LIN {X 0,Y 241.734,Z 622.114,A -85,B 0,C 180,E1 -22159.156,E2 -22159.156} C_VEL
LIN {X 0,Y 239.489,Z 637.629,A -85,B 0,C 180,E1 -22159.816,E2 -22159.816} C_VEL
LIN {X 0,Y 236.435,Z 652.725,A -85,B 0,C 180,E1 -22160.765,E2 -22160.765} C_VEL
LIN {X 0,Y 232.635,Z 667.345,A -85,B 0,C 180,E1 -22162.02,E2 -22162.02} C_VEL
LIN {X 0,Y 228.038,Z 681.642,A -85,B 0,C 180,E1 -22163.62,E2 -22163.62} C_VEL
LIN {X 0,Y 222.936,Z 694.986,A -85,B 0,C 180,E1 -22165.531,E2 -22165.531} C_VEL
LIN {X 0,Y 218.006,Z 706.292,A -85,B 0,C 180,E1 -22167.563,E2 -22167.563} C_VEL
LIN {X 0,Y 212.694,Z 717.163,A -85,B 0,C 180,E1 -22169.995,E2 -22169.995} C_VEL
LIN {X 0,Y 207.139,Z 727.482,A -85,B 0,C 180,E1 -22172.879,E2 -22172.879} C_VEL
LIN {X 0,Y 201.494,Z 737.279,A -85,B 0,C 180,E1 -22176.367,E2 -22176.367} C_VEL
LIN {X 0,Y 196.39,Z 745.451,A -85,B 0,C 180,E1 -22180.103,E2 -22180.103} C_VEL
LIN {X 0,Y 192.203,Z 752.008,A -85,B 0,C 180,E1 -22184.008,E2 -22184.008} C_VEL
LIN {X 0,Y 188.734,Z 757.287,A -85,B 0,C 180,E1 -22188.139,E2 -22188.139} C_VEL
LIN {X 0,Y 185.966,Z 761.59,A -85,B 0,C 180,E1 -22192.797,E2 -22192.797} C_VEL
LIN {X 0,Y 184.093,Z 764.533,A -85,B 0,C 180,E1 -22197.694,E2 -22197.694} C_VEL
LIN {X 0,Y 183.006,Z 766.01,A -85,B 0,C 180,E1 -22202.561,E2 -22202.561} C_VEL
LIN {X 0,Y 182.635,Z 766.103,A -85,B 0,C 180,E1 -22207.452,E2 -22207.452} C_VEL
LIN {X 0,Y 182.792,Z 764.903,A -85,B 0,C 180,E1 -22212.088,E2 -22212.088} C_VEL
LIN {X 0,Y 183.127,Z 763.818,A -85,B 0,C 180,E1 -22214.418,E2 -22214.418} C_VEL
LIN {X 0,Y 184.071,Z 760.704,A -85,B 0,C 180,E1 -22218.996,E2 -22218.996} C_VEL
LIN {X 0,Y 185.74,Z 756.271,A -85,B 0,C 180,E1 -22223.483,E2 -22223.483} C_VEL
LIN {X 0,Y 188.123,Z 750.443,A -85,B 0,C 180,E1 -22227.86,E2 -22227.86} C_VEL
LIN {X 0,Y 191.358,Z 743.051,A -85,B 0,C 180,E1 -22232.106,E2 -22232.106} C_VEL
LIN {X 0,Y 194.901,Z 735.115,A -85,B 0,C 180,E1 -22235.692,E2 -22235.692} C_VEL
LIN {X 0,Y 198.898,Z 726.022,A -85,B 0,C 180,E1 -22238.993,E2 -22238.993} C_VEL
LIN {X 0,Y 203.137,Z 715.83,A -85,B 0,C 180,E1 -22241.982,E2 -22241.982} C_VEL
LIN {X 0,Y 207.665,Z 704.233,A -85,B 0,C 180,E1 -22244.705,E2 -22244.705} C_VEL
LIN {X 0,Y 212.179,Z 691.452,A -85,B 0,C 180,E1 -22247.096,E2 -22247.096} C_VEL
LIN {X 0,Y 216.109,Z 678.872,A -85,B 0,C 180,E1 -22248.979,E2 -22248.979} C_VEL
LIN {X 0,Y 219.617,Z 665.333,A -85,B 0,C 180,E1 -22250.611,E2 -22250.611} C_VEL
LIN {X 0,Y 222.901,Z 650.22,A -85,B 0,C 180,E1 -22251.989,E2 -22251.989} C_VEL
LIN {X 0,Y 225.379,Z 635.225,A -85,B 0,C 180,E1 -22253.003,E2 -22253.003} C_VEL
LIN {X 0,Y 227.257,Z 619.581,A -85,B 0,C 180,E1 -22253.706,E2 -22253.706} C_VEL
LIN {X 0,Y 232.606,Z 539.728,A -85,B 0,C 180,E1 -22256.019,E2 -22256.019} C_VEL
LIN {X 0,Y 229.272,Z 532.768,A -85,B 0,C 180,E1 -22257.137,E2 -22257.137} C_VEL
LIN {X 0,Y 222.382,Z 520.492,A -85,B 0,C 180,E1 -22259.498,E2 -22259.498} C_VEL
LIN {X 0,Y 215.018,Z 508.387,A -85,B 0,C 180,E1 -22262.247,E2 -22262.247} C_VEL
LIN {X 0,Y 206.888,Z 496.398,A -85,B 0,C 180,E1 -22265.594,E2 -22265.594} C_VEL
LIN {X 0,Y 200.691,Z 487.945,A -85,B 0,C 180,E1 -22268.442,E2 -22268.442} C_VEL
LIN {X 0,Y 197.937,Z 484.198,A -85,B 0,C 180,E1 -22269.821,E2 -22269.821} C_VEL
LIN {X 0,Y 194.647,Z 480.304,A -85,B 0,C 180,E1 -22271.528,E2 -22271.528} C_VEL
LIN {X 0,Y 193.678,Z 478.802,A -85,B 0,C 180,E1 -22272.082,E2 -22272.082} C_VEL
LIN {X 0,Y 191.056,Z 476.179,A -85,B 0,C 180,E1 -22273.545,E2 -22273.545} C_VEL
LIN {X 0,Y 189.711,Z 473.644,A -85,B 0,C 180,E1 -22274.429,E2 -22274.429} C_VEL
LIN {X 0,Y 187.18,Z 471.799,A -85,B 0,C 180,E1 -22275.917,E2 -22275.917} C_VEL
LIN {X 0,Y 185.806,Z 469.34,A -85,B 0,C 180,E1 -22276.897,E2 -22276.897} C_VEL
LIN {X 0,Y 185.502,Z 467.989,A -85,B 0,C 180,E1 -22277.235,E2 -22277.235} C_VEL
LIN {X 0,Y 185.52,Z 467.989,A -85,B 0,C 180,E1 -22279.908,E2 -22279.908} C_VEL
LIN {X 0,Y 185.547,Z 467.982,A -85,B 0,C 180,E1 -22282.696,E2 -22282.696} C_VEL
LIN {X 0,Y 185.544,Z 467.991,A -85,B 0,C 180,E1 -22287.974,E2 -22287.974} C_VEL
LIN {X 0,Y 185.584,Z 467.969,A -85,B 0,C 180,E1 -22290.577,E2 -22290.577} C_VEL
LIN {X 0,Y 185.583,Z 467.972,A -85,B 0,C 180,E1 -22295.381,E2 -22295.381} C_VEL
LIN {X 0,Y 185.677,Z 467.972,A -85,B 0,C 180,E1 -22301.133,E2 -22301.133} C_VEL
LIN {X 0,Y 185.768,Z 467.969,A -85,B 0,C 180,E1 -22306.879,E2 -22306.879} C_VEL
LIN {X 0,Y 186.017,Z 467.914,A -85,B 0,C 180,E1 -22311.307,E2 -22311.307} C_VEL
LIN {X 0,Y 186.21,Z 467.89,A -85,B 0,C 180,E1 -22317.836,E2 -22317.836} C_VEL
LIN {X 0,Y 186.409,Z 467.888,A -85,B 0,C 180,E1 -22319.999,E2 -22319.999} C_VEL
LIN {X 0,Y 185.926,Z 467.912,A -85,B 0,C 180,E1 -22324.335,E2 -22324.335} C_VEL
LIN {X 0,Y 186.016,Z 467.939,A -85,B 0,C 180,E1 -22328.692,E2 -22328.692} C_VEL
LIN {X 0,Y 185.737,Z 467.946,A -85,B 0,C 180,E1 -22333.122,E2 -22333.122} C_VEL
LIN {X 0,Y 185.72,Z 467.953,A -85,B 0,C 180,E1 -22337.621,E2 -22337.621} C_VEL
LIN {X 0,Y 185.652,Z 468.142,A -85,B 0,C 180,E1 -22340.497,E2 -22340.497} C_VEL
LIN {X 0,Y 186.512,Z 470.625,A -85,B 0,C 180,E1 -22341.192,E2 -22341.192} C_VEL
LIN {X 0,Y 188.316,Z 472.728,A -85,B 0,C 180,E1 -22342.346,E2 -22342.346} C_VEL
LIN {X 0,Y 190.035,Z 473.955,A -85,B 0,C 180,E1 -22343.353,E2 -22343.353} C_VEL
LIN {X 0,Y 191.815,Z 477.044,A -85,B 0,C 180,E1 -22344.486,E2 -22344.486} C_VEL
LIN {X 0,Y 194.264,Z 479.432,A -85,B 0,C 180,E1 -22345.825,E2 -22345.825} C_VEL
LIN {X 0,Y 196.595,Z 482.776,A -85,B 0,C 180,E1 -22347.098,E2 -22347.098} C_VEL
LIN {X 0,Y 198.231,Z 484.658,A -85,B 0,C 180,E1 -22347.919,E2 -22347.919} C_VEL
LIN {X 0,Y 201.912,Z 489.596,A -85,B 0,C 180,E1 -22349.729,E2 -22349.729} C_VEL
LIN {X 0,Y 206.916,Z 496.507,A -85,B 0,C 180,E1 -22352.012,E2 -22352.012} C_VEL
LIN {X 0,Y 213.331,Z 507.607,A -85,B 0,C 180,E1 -22354.774,E2 -22354.774} C_VEL
LIN {X 0,Y 220.542,Z 521.142,A -85,B 0,C 180,E1 -22357.615,E2 -22357.615} C_VEL
LIN {X 0,Y 227.101,Z 535.188,A -85,B 0,C 180,E1 -22360.024,E2 -22360.024} C_VEL
LIN {X 0,Y 231.364,Z 545.348,A -85,B 0,C 180,E1 -22361.526,E2 -22361.526} C_VEL
LIN {X 0,Y 231.715,Z 547.693,A -85,B 0,C 180,E1 -22361.713,E2 -22361.713} C_VEL
LIN {X 0,Y 231.08,Z 551.504,A -85,B 0,C 180,E1 -22361.731,E2 -22361.731} C_VEL
LIN {X 0,Y 229.684,Z 555.211,A -85,B 0,C 180,E1 -22361.564,E2 -22361.564} C_VEL
LIN {X 0,Y 226.875,Z 561.739,A -85,B 0,C 180,E1 -22361.18,E2 -22361.18} C_VEL
LIN {X 0,Y 225.979,Z 565.9,A -85,B 0,C 180,E1 -22361.151,E2 -22361.151} C_VEL
LIN {X 0,Y 221.35,Z 631.555,A -85,B 0,C 180,E1 -22363.091,E2 -22363.091} C_VEL
LIN {X 0,Y 219.258,Z 647.344,A -85,B 0,C 180,E1 -22363.845,E2 -22363.845} C_VEL
LIN {X 0,Y 216.358,Z 662.488,A -85,B 0,C 180,E1 -22364.883,E2 -22364.883} C_VEL
LIN {X 0,Y 213.032,Z 676.219,A -85,B 0,C 180,E1 -22366.147,E2 -22366.147} C_VEL
LIN {X 0,Y 209.192,Z 689.735,A -85,B 0,C 180,E1 -22367.784,E2 -22367.784} C_VEL
LIN {X 0,Y 204.553,Z 703.482,A -85,B 0,C 180,E1 -22369.893,E2 -22369.893} C_VEL
LIN {X 0,Y 199.88,Z 715.958,A -85,B 0,C 180,E1 -22372.343,E2 -22372.343} C_VEL
LIN {X 0,Y 194.715,Z 728.142,A -85,B 0,C 180,E1 -22375.355,E2 -22375.355} C_VEL
LIN {X 0,Y 190.501,Z 737.849,A -85,B 0,C 180,E1 -22378.384,E2 -22378.384} C_VEL
LIN {X 0,Y 186.487,Z 746.873,A -85,B 0,C 180,E1 -22381.895,E2 -22381.895} C_VEL
LIN {X 0,Y 182.942,Z 754.535,A -85,B 0,C 180,E1 -22385.607,E2 -22385.607} C_VEL
LIN {X 0,Y 180.179,Z 760.857,A -85,B 0,C 180,E1 -22389.447,E2 -22389.447} C_VEL
LIN {X 0,Y 177.951,Z 766.646,A -85,B 0,C 180,E1 -22393.95,E2 -22393.95} C_VEL
LIN {X 0,Y 176.573,Z 771.032,A -85,B 0,C 180,E1 -22398.52,E2 -22398.52} C_VEL
LIN {X 0,Y 176.011,Z 774.126,A -85,B 0,C 180,E1 -22403.119,E2 -22403.119} C_VEL
LIN {X 0,Y 175.948,Z 775.99,A -85,B 0,C 180,E1 -22407.71,E2 -22407.71} C_VEL
LIN {X 0,Y 176.088,Z 776.458,A -85,B 0,C 180,E1 -22409.999,E2 -22409.999} C_VEL
LIN {X 0,Y 175.93,Z 776.478,A -85,B 0,C 180,E1 -22414.581,E2 -22414.581} C_VEL
LIN {X 0,Y 176.219,Z 775.363,A -85,B 0,C 180,E1 -22419.178,E2 -22419.178} C_VEL
LIN {X 0,Y 177.172,Z 773.116,A -85,B 0,C 180,E1 -22423.767,E2 -22423.767} C_VEL
LIN {X 0,Y 179.099,Z 769.707,A -85,B 0,C 180,E1 -22428.294,E2 -22428.294} C_VEL
LIN {X 0,Y 181.995,Z 765.027,A -85,B 0,C 180,E1 -22432.714,E2 -22432.714} C_VEL
LIN {X 0,Y 185.858,Z 758.973,A -85,B 0,C 180,E1 -22436.984,E2 -22436.984} C_VEL
LIN {X 0,Y 190.198,Z 752.43,A -85,B 0,C 180,E1 -22440.534,E2 -22440.534} C_VEL
LIN {X 0,Y 195.326,Z 743.996,A -85,B 0,C 180,E1 -22444.217,E2 -22444.217} C_VEL
LIN {X 0,Y 200.526,Z 735.309,A -85,B 0,C 180,E1 -22447.196,E2 -22447.196} C_VEL
LIN {X 0,Y 206.805,Z 724.104,A -85,B 0,C 180,E1 -22450.216,E2 -22450.216} C_VEL
LIN {X 0,Y 212.592,Z 712.612,A -85,B 0,C 180,E1 -22452.662,E2 -22452.662} C_VEL
LIN {X 0,Y 218.333,Z 699.772,A -85,B 0,C 180,E1 -22454.817,E2 -22454.817} C_VEL
LIN {X 0,Y 223.651,Z 686.095,A -85,B 0,C 180,E1 -22456.606,E2 -22456.606} C_VEL
LIN {X 0,Y 228.157,Z 672.417,A -85,B 0,C 180,E1 -22457.997,E2 -22457.997} C_VEL
LIN {X 0,Y 231.692,Z 659.718,A -85,B 0,C 180,E1 -22458.983,E2 -22458.983} C_VEL
LIN {X 0,Y 235.025,Z 644.454,A -85,B 0,C 180,E1 -22459.851,E2 -22459.851} C_VEL
LIN {X 0,Y 237.229,Z 629.636,A -85,B 0,C 180,E1 -22460.465,E2 -22460.465} C_VEL
LIN {X 0,Y 243.268,Z 558.028,A -85,B 0,C 180,E1 -22462.41,E2 -22462.41} C_VEL
LIN {X 0,Y 241.558,Z 553.044,A -85,B 0,C 180,E1 -22463.369,E2 -22463.369} C_VEL
LIN {X 0,Y 237.978,Z 544.448,A -85,B 0,C 180,E1 -22465.447,E2 -22465.447} C_VEL
LIN {X 0,Y 234.157,Z 536.255,A -85,B 0,C 180,E1 -22467.872,E2 -22467.872} C_VEL
LIN {X 0,Y 230.657,Z 529.337,A -85,B 0,C 180,E1 -22470.376,E2 -22470.376} C_VEL
LIN {X 0,Y 228.094,Z 524.709,A -85,B 0,C 180,E1 -22472.473,E2 -22472.473} C_VEL
LIN {X 0,Y 225.797,Z 520.619,A -85,B 0,C 180,E1 -22474.627,E2 -22474.627} C_VEL
LIN {X 0,Y 223.343,Z 517.052,A -85,B 0,C 180,E1 -22477.295,E2 -22477.295} C_VEL
LIN {X 0,Y 222.418,Z 516.005,A -85,B 0,C 180,E1 -22478.45,E2 -22478.45} C_VEL
LIN {X 0,Y 220.305,Z 512.836,A -85,B 0,C 180,E1 -22481.921,E2 -22481.921} C_VEL
LIN {X 0,Y 219.775,Z 511.515,A -85,B 0,C 180,E1 -22483.274,E2 -22483.274} C_VEL
LIN {X 0,Y 218.477,Z 510.721,A -85,B 0,C 180,E1 -22488.872,E2 -22488.872} C_VEL
LIN {X 0,Y 219.031,Z 510.958,A -85,B 0,C 180,E1 -22493.09,E2 -22493.09} C_VEL
LIN {X 0,Y 220.41,Z 511.803,A -85,B 0,C 180,E1 -22496.486,E2 -22496.486} C_VEL
LIN {X 0,Y 222.476,Z 515.52,A -85,B 0,C 180,E1 -22500,E2 -22500} C_VEL
LIN {X 0,Y 223.564,Z 516.901,A -85,B 0,C 180,E1 -22501.369,E2 -22501.369} C_VEL
LIN {X 0,Y 226.489,Z 521.275,A -85,B 0,C 180,E1 -22504.464,E2 -22504.464} C_VEL
LIN {X 0,Y 229.47,Z 526.02,A -85,B 0,C 180,E1 -22507.037,E2 -22507.037} C_VEL
LIN {X 0,Y 232.882,Z 531.325,A -85,B 0,C 180,E1 -22509.526,E2 -22509.526} C_VEL
LIN {X 0,Y 237.163,Z 538.709,A -85,B 0,C 180,E1 -22512.255,E2 -22512.255} C_VEL
LIN {X 0,Y 242.095,Z 547.889,A -85,B 0,C 180,E1 -22514.992,E2 -22514.992} C_VEL
LIN {X 0,Y 243.679,Z 551.454,A -85,B 0,C 180,E1 -22515.825,E2 -22515.825} C_VEL
LIN {X 0,Y 237.763,Z 621.792,A -85,B 0,C 180,E1 -22517.744,E2 -22517.744} C_VEL
LIN {X 0,Y 235.49,Z 637.313,A -85,B 0,C 180,E1 -22518.392,E2 -22518.392} C_VEL
LIN {X 0,Y 232.244,Z 652.905,A -85,B 0,C 180,E1 -22519.362,E2 -22519.362} C_VEL
LIN {X 0,Y 228.145,Z 667.998,A -85,B 0,C 180,E1 -22520.663,E2 -22520.663} C_VEL
LIN {X 0,Y 223.752,Z 681.221,A -85,B 0,C 180,E1 -22522.143,E2 -22522.143} C_VEL
LIN {X 0,Y 218.408,Z 694.763,A -85,B 0,C 180,E1 -22524.072,E2 -22524.072} C_VEL
LIN {X 0,Y 213.217,Z 706.192,A -85,B 0,C 180,E1 -22526.121,E2 -22526.121} C_VEL
LIN {X 0,Y 207.861,Z 716.722,A -85,B 0,C 180,E1 -22528.471,E2 -22528.471} C_VEL
LIN {X 0,Y 201.824,Z 727.5,A -85,B 0,C 180,E1 -22531.49,E2 -22531.49} C_VEL
LIN {X 0,Y 196.463,Z 736.323,A -85,B 0,C 180,E1 -22534.64,E2 -22534.64} C_VEL
LIN {X 0,Y 191.661,Z 743.7,A -85,B 0,C 180,E1 -22537.935,E2 -22537.935} C_VEL
LIN {X 0,Y 187.467,Z 749.95,A -85,B 0,C 180,E1 -22541.431,E2 -22541.431} C_VEL
LIN {X 0,Y 183.952,Z 755.015,A -85,B 0,C 180,E1 -22545.027,E2 -22545.027} C_VEL
LIN {X 0,Y 180.326,Z 760.213,A -85,B 0,C 180,E1 -22549.981,E2 -22549.981} C_VEL
LIN {X 0,Y 178.38,Z 762.986,A -85,B 0,C 180,E1 -22553.775,E2 -22553.775} C_VEL
LIN {X 0,Y 176.639,Z 765.401,A -85,B 0,C 180,E1 -22558.855,E2 -22558.855} C_VEL
LIN {X 0,Y 175.71,Z 766.396,A -85,B 0,C 180,E1 -22563.9,E2 -22563.9} C_VEL
LIN {X 0,Y 175.528,Z 766.041,A -85,B 0,C 180,E1 -22568.88,E2 -22568.88} C_VEL
LIN {X 0,Y 175.898,Z 764.397,A -85,B 0,C 180,E1 -22573.76,E2 -22573.76} C_VEL
LIN {X 0,Y 176.826,Z 761.484,A -85,B 0,C 180,E1 -22578.539,E2 -22578.539} C_VEL
LIN {X 0,Y 178.464,Z 757.262,A -85,B 0,C 180,E1 -22583.216,E2 -22583.216} C_VEL
LIN {X 0,Y 180.846,Z 751.658,A -85,B 0,C 180,E1 -22587.774,E2 -22587.774} C_VEL
LIN {X 0,Y 184.124,Z 744.508,A -85,B 0,C 180,E1 -22592.189,E2 -22592.189} C_VEL
LIN {X 0,Y 187.675,Z 736.853,A -85,B 0,C 180,E1 -22595.912,E2 -22595.912} C_VEL
LIN {X 0,Y 192.068,Z 727.393,A -85,B 0,C 180,E1 -22599.549,E2 -22599.549} C_VEL
LIN {X 0,Y 196.845,Z 716.415,A -85,B 0,C 180,E1 -22602.895,E2 -22602.895} C_VEL
LIN {X 0,Y 201.511,Z 704.901,A -85,B 0,C 180,E1 -22605.683,E2 -22605.683} C_VEL
LIN {X 0,Y 206.186,Z 692.282,A -85,B 0,C 180,E1 -22608.105,E2 -22608.105} C_VEL
LIN {X 0,Y 210.248,Z 679.75,A -85,B 0,C 180,E1 -22610.038,E2 -22610.038} C_VEL
LIN {X 0,Y 213.892,Z 666.336,A -85,B 0,C 180,E1 -22611.695,E2 -22611.695} C_VEL
LIN {X 0,Y 217.262,Z 651.491,A -85,B 0,C 180,E1 -22613.094,E2 -22613.094} C_VEL
LIN {X 0,Y 219.947,Z 636.009,A -85,B 0,C 180,E1 -22614.168,E2 -22614.168} C_VEL
LIN {X 0,Y 221.826,Z 621.311,A -85,B 0,C 180,E1 -22614.858,E2 -22614.858} C_VEL
LIN {X 0,Y 227.367,Z 542.121,A -85,B 0,C 180,E1 -22617.179,E2 -22617.179} C_VEL
LIN {X 0,Y 221.677,Z 531.086,A -85,B 0,C 180,E1 -22619.174,E2 -22619.174} C_VEL
LIN {X 0,Y 212.987,Z 516.086,A -85,B 0,C 180,E1 -22622.465,E2 -22622.465} C_VEL
LIN {X 0,Y 205.507,Z 504.756,A -85,B 0,C 180,E1 -22625.595,E2 -22625.595} C_VEL
LIN {X 0,Y 200.107,Z 497.094,A -85,B 0,C 180,E1 -22628.09,E2 -22628.09} C_VEL
LIN {X 0,Y 197.355,Z 493.344,A -85,B 0,C 180,E1 -22629.459,E2 -22629.459} C_VEL
LIN {X 0,Y 194.47,Z 489.422,A -85,B 0,C 180,E1 -22630.968,E2 -22630.968} C_VEL
LIN {X 0,Y 191.496,Z 485.498,A -85,B 0,C 180,E1 -22632.629,E2 -22632.629} C_VEL
LIN {X 0,Y 188.184,Z 481.692,A -85,B 0,C 180,E1 -22634.588,E2 -22634.588} C_VEL
LIN {X 0,Y 186.961,Z 479.881,A -85,B 0,C 180,E1 -22635.378,E2 -22635.378} C_VEL
LIN {X 0,Y 184.461,Z 477.453,A -85,B 0,C 180,E1 -22636.981,E2 -22636.981} C_VEL
LIN {X 0,Y 182.959,Z 474.622,A -85,B 0,C 180,E1 -22638.13,E2 -22638.13} C_VEL
LIN {X 0,Y 180.327,Z 472.837,A -85,B 0,C 180,E1 -22639.978,E2 -22639.978} C_VEL
LIN {X 0,Y 178.868,Z 470.544,A -85,B 0,C 180,E1 -22641.2,E2 -22641.2} C_VEL
LIN {X 0,Y 178.466,Z 468.876,A -85,B 0,C 180,E1 -22641.703,E2 -22641.703} C_VEL
LIN {X 0,Y 178.492,Z 468.874,A -85,B 0,C 180,E1 -22646.547,E2 -22646.547} C_VEL
LIN {X 0,Y 178.525,Z 468.848,A -85,B 0,C 180,E1 -22650.007,E2 -22650.007} C_VEL
LIN {X 0,Y 178.523,Z 468.856,A -85,B 0,C 180,E1 -22654.886,E2 -22654.886} C_VEL
LIN {X 0,Y 178.625,Z 468.854,A -85,B 0,C 180,E1 -22660.785,E2 -22660.785} C_VEL
LIN {X 0,Y 178.685,Z 468.849,A -85,B 0,C 180,E1 -22666.349,E2 -22666.349} C_VEL
LIN {X 0,Y 178.966,Z 468.79,A -85,B 0,C 180,E1 -22670.962,E2 -22670.962} C_VEL
LIN {X 0,Y 179.156,Z 468.767,A -85,B 0,C 180,E1 -22677.751,E2 -22677.751} C_VEL
LIN {X 0,Y 179.372,Z 468.764,A -85,B 0,C 180,E1 -22679.999,E2 -22679.999} C_VEL
LIN {X 0,Y 178.874,Z 468.79,A -85,B 0,C 180,E1 -22684.506,E2 -22684.506} C_VEL
LIN {X 0,Y 178.966,Z 468.813,A -85,B 0,C 180,E1 -22689.037,E2 -22689.037} C_VEL
LIN {X 0,Y 178.67,Z 468.831,A -85,B 0,C 180,E1 -22693.651,E2 -22693.651} C_VEL
LIN {X 0,Y 178.66,Z 468.886,A -85,B 0,C 180,E1 -22696.056,E2 -22696.056} C_VEL
LIN {X 0,Y 179.368,Z 471.182,A -85,B 0,C 180,E1 -22696.796,E2 -22696.796} C_VEL
LIN {X 0,Y 181.346,Z 473.561,A -85,B 0,C 180,E1 -22698.357,E2 -22698.357} C_VEL
LIN {X 0,Y 183.205,Z 474.802,A -85,B 0,C 180,E1 -22699.631,E2 -22699.631} C_VEL
LIN {X 0,Y 184.787,Z 477.743,A -85,B 0,C 180,E1 -22700.816,E2 -22700.816} C_VEL
LIN {X 0,Y 187.588,Z 480.382,A -85,B 0,C 180,E1 -22702.571,E2 -22702.571} C_VEL
LIN {X 0,Y 189.993,Z 483.914,A -85,B 0,C 180,E1 -22704.1,E2 -22704.1} C_VEL
LIN {X 0,Y 191.71,Z 485.705,A -85,B 0,C 180,E1 -22705.077,E2 -22705.077} C_VEL
LIN {X 0,Y 194.528,Z 489.448,A -85,B 0,C 180,E1 -22706.647,E2 -22706.647} C_VEL
LIN {X 0,Y 199.16,Z 495.74,A -85,B 0,C 180,E1 -22709.026,E2 -22709.026} C_VEL
LIN {X 0,Y 203.688,Z 502.029,A -85,B 0,C 180,E1 -22711.168,E2 -22711.168} C_VEL
LIN {X 0,Y 211.32,Z 515.671,A -85,B 0,C 180,E1 -22714.573,E2 -22714.573} C_VEL
LIN {X 0,Y 217.721,Z 528.372,A -85,B 0,C 180,E1 -22717.173,E2 -22717.173} C_VEL
LIN {X 0,Y 224.288,Z 543.054,A -85,B 0,C 180,E1 -22719.675,E2 -22719.675} C_VEL
LIN {X 0,Y 227.042,Z 550.077,A -85,B 0,C 180,E1 -22720.69,E2 -22720.69} C_VEL
LIN {X 0,Y 225.979,Z 565.9,A -85,B 0,C 180,E1 -22721.151,E2 -22721.151} C_VEL
LIN {X 0,Y 225.101,Z 571.739,A -85,B 0,C 180,E1 -22721.204,E2 -22721.204} C_VEL
LIN {X 0,Y 219.653,Z 590.729,A -85,B 0,C 180,E1 -22720.734,E2 -22720.734} C_VEL
LIN {X 0,Y 218.743,Z 596.569,A -85,B 0,C 180,E1 -22720.779,E2 -22720.779} C_VEL
LIN {X 0,Y 216.099,Z 631.564,A -85,B 0,C 180,E1 -22721.844,E2 -22721.844} C_VEL
LIN {X 0,Y 213.948,Z 647.286,A -85,B 0,C 180,E1 -22722.605,E2 -22722.605} C_VEL
LIN {X 0,Y 211.081,Z 661.823,A -85,B 0,C 180,E1 -22723.599,E2 -22723.599} C_VEL
LIN {X 0,Y 207.356,Z 676.746,A -85,B 0,C 180,E1 -22725,E2 -22725} C_VEL
LIN {X 0,Y 203.517,Z 689.744,A -85,B 0,C 180,E1 -22726.6,E2 -22726.6} C_VEL
LIN {X 0,Y 198.649,Z 703.658,A -85,B 0,C 180,E1 -22728.781,E2 -22728.781} C_VEL
LIN {X 0,Y 193.814,Z 716.078,A -85,B 0,C 180,E1 -22731.279,E2 -22731.279} C_VEL
LIN {X 0,Y 188.845,Z 727.381,A -85,B 0,C 180,E1 -22734.115,E2 -22734.115} C_VEL
LIN {X 0,Y 184.524,Z 736.717,A -85,B 0,C 180,E1 -22737.052,E2 -22737.052} C_VEL
LIN {X 0,Y 180.796,Z 745.008,A -85,B 0,C 180,E1 -22740.288,E2 -22740.288} C_VEL
LIN {X 0,Y 176.882,Z 752.971,A -85,B 0,C 180,E1 -22744.082,E2 -22744.082} C_VEL
LIN {X 0,Y 173.452,Z 760.391,A -85,B 0,C 180,E1 -22748.612,E2 -22748.612} C_VEL
LIN {X 0,Y 171.074,Z 766.242,A -85,B 0,C 180,E1 -22753.286,E2 -22753.286} C_VEL
LIN {X 0,Y 169.569,Z 770.683,A -85,B 0,C 180,E1 -22758.039,E2 -22758.039} C_VEL
LIN {X 0,Y 168.93,Z 773.83,A -85,B 0,C 180,E1 -22762.829,E2 -22762.829} C_VEL
LIN {X 0,Y 168.857,Z 775.732,A -85,B 0,C 180,E1 -22767.613,E2 -22767.613} C_VEL
LIN {X 0,Y 168.996,Z 776.213,A -85,B 0,C 180,E1 -22769.999,E2 -22769.999} C_VEL
LIN {X 0,Y 168.845,Z 776.282,A -85,B 0,C 180,E1 -22774.774,E2 -22774.774} C_VEL
LIN {X 0,Y 169.158,Z 775.22,A -85,B 0,C 180,E1 -22779.565,E2 -22779.565} C_VEL
LIN {X 0,Y 170.221,Z 773.029,A -85,B 0,C 180,E1 -22784.341,E2 -22784.341} C_VEL
LIN {X 0,Y 172.317,Z 769.67,A -85,B 0,C 180,E1 -22789.042,E2 -22789.042} C_VEL
LIN {X 0,Y 175.414,Z 765.026,A -85,B 0,C 180,E1 -22793.617,E2 -22793.617} C_VEL
LIN {X 0,Y 179.519,Z 759.048,A -85,B 0,C 180,E1 -22798.019,E2 -22798.019} C_VEL
LIN {X 0,Y 184.762,Z 751.584,A -85,B 0,C 180,E1 -22802.175,E2 -22802.175} C_VEL
LIN {X 0,Y 190.014,Z 743.452,A -85,B 0,C 180,E1 -22805.733,E2 -22805.733} C_VEL
LIN {X 0,Y 195.813,Z 734.172,A -85,B 0,C 180,E1 -22808.908,E2 -22808.908} C_VEL
LIN {X 0,Y 201.459,Z 724.554,A -85,B 0,C 180,E1 -22811.514,E2 -22811.514} C_VEL
LIN {X 0,Y 207.455,Z 713.229,A -85,B 0,C 180,E1 -22813.984,E2 -22813.984} C_VEL
LIN {X 0,Y 213.354,Z 700.704,A -85,B 0,C 180,E1 -22816.134,E2 -22816.134} C_VEL
LIN {X 0,Y 218.886,Z 687.172,A -85,B 0,C 180,E1 -22817.942,E2 -22817.942} C_VEL
LIN {X 0,Y 223.521,Z 673.816,A -85,B 0,C 180,E1 -22819.334,E2 -22819.334} C_VEL
LIN {X 0,Y 227.466,Z 660.311,A -85,B 0,C 180,E1 -22820.396,E2 -22820.396} C_VEL
LIN {X 0,Y 231.045,Z 644.523,A -85,B 0,C 180,E1 -22821.297,E2 -22821.297} C_VEL
LIN {X 0,Y 233.41,Z 629.037,A -85,B 0,C 180,E1 -22821.929,E2 -22821.929} C_VEL
LIN {X 0,Y 239.383,Z 561.006,A -85,B 0,C 180,E1 -22823.769,E2 -22823.769} C_VEL
LIN {X 0,Y 238.903,Z 559.062,A -85,B 0,C 180,E1 -22824.093,E2 -22824.093} C_VEL
LIN {X 0,Y 235.248,Z 549.883,A -85,B 0,C 180,E1 -22826.335,E2 -22826.335} C_VEL
LIN {X 0,Y 231.652,Z 541.788,A -85,B 0,C 180,E1 -22828.788,E2 -22828.788} C_VEL
LIN {X 0,Y 228.565,Z 535.35,A -85,B 0,C 180,E1 -22831.162,E2 -22831.162} C_VEL
LIN {X 0,Y 226.277,Z 531.044,A -85,B 0,C 180,E1 -22833.141,E2 -22833.141} C_VEL
LIN {X 0,Y 224.362,Z 527.366,A -85,B 0,C 180,E1 -22835.057,E2 -22835.057} C_VEL
LIN {X 0,Y 221.879,Z 523.581,A -85,B 0,C 180,E1 -22837.906,E2 -22837.906} C_VEL
LIN {X 0,Y 219.223,Z 519.836,A -85,B 0,C 180,E1 -22842.194,E2 -22842.194} C_VEL
LIN {X 0,Y 218.753,Z 518.515,A -85,B 0,C 180,E1 -22843.488,E2 -22843.488} C_VEL
LIN {X 0,Y 217.555,Z 517.765,A -85,B 0,C 180,E1 -22848.824,E2 -22848.824} C_VEL
LIN {X 0,Y 218.06,Z 517.969,A -85,B 0,C 180,E1 -22852.933,E2 -22852.933} C_VEL
LIN {X 0,Y 219.307,Z 518.765,A -85,B 0,C 180,E1 -22856.156,E2 -22856.156} C_VEL
LIN {X 0,Y 221.273,Z 522.4,A -85,B 0,C 180,E1 -22859.671,E2 -22859.671} C_VEL
LIN {X 0,Y 222.261,Z 523.81,A -85,B 0,C 180,E1 -22861.001,E2 -22861.001} C_VEL
LIN {X 0,Y 224.909,Z 527.891,A -85,B 0,C 180,E1 -22863.923,E2 -22863.923} C_VEL
LIN {X 0,Y 227.68,Z 532.492,A -85,B 0,C 180,E1 -22866.447,E2 -22866.447} C_VEL
LIN {X 0,Y 231.04,Z 537.931,A -85,B 0,C 180,E1 -22869.025,E2 -22869.025} C_VEL
LIN {X 0,Y 235.185,Z 545.538,A -85,B 0,C 180,E1 -22871.792,E2 -22871.792} C_VEL
LIN {X 0,Y 239.421,Z 553.702,A -85,B 0,C 180,E1 -22874.245,E2 -22874.245} C_VEL
LIN {X 0,Y 239.784,Z 554.786,A -85,B 0,C 180,E1 -22874.467,E2 -22874.467} C_VEL
LIN {X 0,Y 233.778,Z 623.026,A -85,B 0,C 180,E1 -22876.336,E2 -22876.336} C_VEL
LIN {X 0,Y 231.281,Z 638.916,A -85,B 0,C 180,E1 -22877.016,E2 -22877.016} C_VEL
LIN {X 0,Y 228.067,Z 653.628,A -85,B 0,C 180,E1 -22877.949,E2 -22877.949} C_VEL
LIN {X 0,Y 224.115,Z 667.784,A -85,B 0,C 180,E1 -22879.168,E2 -22879.168} C_VEL
LIN {X 0,Y 219.662,Z 680.779,A -85,B 0,C 180,E1 -22880.607,E2 -22880.607} C_VEL
LIN {X 0,Y 214.023,Z 694.624,A -85,B 0,C 180,E1 -22882.553,E2 -22882.553} C_VEL
LIN {X 0,Y 208.088,Z 707.146,A -85,B 0,C 180,E1 -22884.817,E2 -22884.817} C_VEL
LIN {X 0,Y 201.948,Z 718.586,A -85,B 0,C 180,E1 -22887.452,E2 -22887.452} C_VEL
LIN {X 0,Y 195.752,Z 728.995,A -85,B 0,C 180,E1 -22890.5,E2 -22890.5} C_VEL
LIN {X 0,Y 190.317,Z 737.419,A -85,B 0,C 180,E1 -22893.637,E2 -22893.637} C_VEL
LIN {X 0,Y 184.654,Z 745.601,A -85,B 0,C 180,E1 -22897.516,E2 -22897.516} C_VEL
LIN {X 0,Y 179.519,Z 752.684,A -85,B 0,C 180,E1 -22901.944,E2 -22901.944} C_VEL
LIN {X 0,Y 175.857,Z 757.537,A -85,B 0,C 180,E1 -22906.002,E2 -22906.002} C_VEL
LIN {X 0,Y 172.77,Z 761.619,A -85,B 0,C 180,E1 -22910.615,E2 -22910.615} C_VEL
LIN {X 0,Y 170.557,Z 764.534,A -85,B 0,C 180,E1 -22915.501,E2 -22915.501} C_VEL
LIN {X 0,Y 169.079,Z 766.265,A -85,B 0,C 180,E1 -22920.798,E2 -22920.798} C_VEL
LIN {X 0,Y 168.49,Z 766.656,A -85,B 0,C 180,E1 -22925.349,E2 -22925.349} C_VEL
LIN {X 0,Y 168.46,Z 765.853,A -85,B 0,C 180,E1 -22930.505,E2 -22930.505} C_VEL
LIN {X 0,Y 169.077,Z 763.761,A -85,B 0,C 180,E1 -22935.559,E2 -22935.559} C_VEL
LIN {X 0,Y 170.32,Z 760.376,A -85,B 0,C 180,E1 -22940.501,E2 -22940.501} C_VEL
LIN {X 0,Y 172.274,Z 755.672,A -85,B 0,C 180,E1 -22945.321,E2 -22945.321} C_VEL
LIN {X 0,Y 175.123,Z 749.542,A -85,B 0,C 180,E1 -22950.001,E2 -22950.001} C_VEL
LIN {X 0,Y 178.89,Z 741.818,A -85,B 0,C 180,E1 -22954.508,E2 -22954.508} C_VEL
LIN {X 0,Y 182.88,Z 733.529,A -85,B 0,C 180,E1 -22958.287,E2 -22958.287} C_VEL
LIN {X 0,Y 186.919,Z 725.063,A -85,B 0,C 180,E1 -22961.386,E2 -22961.386} C_VEL
LIN {X 0,Y 191.382,Z 715.139,A -85,B 0,C 180,E1 -22964.353,E2 -22964.353} C_VEL
LIN {X 0,Y 196.267,Z 703.334,A -85,B 0,C 180,E1 -22967.184,E2 -22967.184} C_VEL
LIN {X 0,Y 200.913,Z 691.046,A -85,B 0,C 180,E1 -22969.516,E2 -22969.516} C_VEL
LIN {X 0,Y 205.374,Z 677.352,A -85,B 0,C 180,E1 -22971.585,E2 -22971.585} C_VEL
LIN {X 0,Y 209.233,Z 663.26,A -85,B 0,C 180,E1 -22973.247,E2 -22973.247} C_VEL
LIN {X 0,Y 212.461,Z 648.73,A -85,B 0,C 180,E1 -22974.555,E2 -22974.555} C_VEL
LIN {X 0,Y 214.973,Z 633.905,A -85,B 0,C 180,E1 -22975.54,E2 -22975.54} C_VEL
LIN {X 0,Y 216.845,Z 618.668,A -85,B 0,C 180,E1 -22976.206,E2 -22976.206} C_VEL
LIN {X 0,Y 222.171,Z 544.527,A -85,B 0,C 180,E1 -22978.394,E2 -22978.394} C_VEL
LIN {X 0,Y 215.545,Z 532.003,A -85,B 0,C 180,E1 -22980.862,E2 -22980.862} C_VEL
LIN {X 0,Y 207.705,Z 518.615,A -85,B 0,C 180,E1 -22984.038,E2 -22984.038} C_VEL
LIN {X 0,Y 200.433,Z 507.51,A -85,B 0,C 180,E1 -22987.304,E2 -22987.304} C_VEL
LIN {X 0,Y 194.584,Z 499.285,A -85,B 0,C 180,E1 -22990.238,E2 -22990.238} C_VEL
LIN {X 0,Y 191.429,Z 495.084,A -85,B 0,C 180,E1 -22991.958,E2 -22991.958} C_VEL
LIN {X 0,Y 188.183,Z 490.812,A -85,B 0,C 180,E1 -22993.876,E2 -22993.876} C_VEL
LIN {X 0,Y 185.379,Z 487.256,A -85,B 0,C 180,E1 -22995.637,E2 -22995.637} C_VEL
LIN {X 0,Y 184.608,Z 486.183,A -85,B 0,C 180,E1 -22996.154,E2 -22996.154} C_VEL
LIN {X 0,Y 182.112,Z 483.563,A -85,B 0,C 180,E1 -22997.845,E2 -22997.845} C_VEL
LIN {X 0,Y 180.723,Z 481.153,A -85,B 0,C 180,E1 -22998.939,E2 -22998.939} C_VEL
LIN {X 0,Y 177.885,Z 478.745,A -85,B 0,C 180,E1 -23001.063,E2 -23001.063} C_VEL
LIN {X 0,Y 176.376,Z 475.89,A -85,B 0,C 180,E1 -23002.464,E2 -23002.464} C_VEL
LIN {X 0,Y 173.129,Z 473.525,A -85,B 0,C 180,E1 -23005.366,E2 -23005.366} C_VEL
LIN {X 0,Y 171.755,Z 471.189,A -85,B 0,C 180,E1 -23006.906,E2 -23006.906} C_VEL
LIN {X 0,Y 171.401,Z 469.758,A -85,B 0,C 180,E1 -23007.44,E2 -23007.44} C_VEL
LIN {X 0,Y 171.45,Z 469.729,A -85,B 0,C 180,E1 -23010.534,E2 -23010.534} C_VEL
LIN {X 0,Y 171.448,Z 469.729,A -85,B 0,C 180,E1 -23015.8,E2 -23015.8} C_VEL
LIN {X 0,Y 171.581,Z 469.73,A -85,B 0,C 180,E1 -23020.871,E2 -23020.871} C_VEL
LIN {X 0,Y 171.597,Z 469.724,A -85,B 0,C 180,E1 -23025.774,E2 -23025.774} C_VEL
LIN {X 0,Y 171.894,Z 469.669,A -85,B 0,C 180,E1 -23030.587,E2 -23030.587} C_VEL
LIN {X 0,Y 171.824,Z 469.69,A -85,B 0,C 180,E1 -23035.307,E2 -23035.307} C_VEL
LIN {X 0,Y 172.335,Z 469.641,A -85,B 0,C 180,E1 -23039.999,E2 -23039.999} C_VEL
LIN {X 0,Y 171.823,Z 469.668,A -85,B 0,C 180,E1 -23044.692,E2 -23044.692} C_VEL
LIN {X 0,Y 171.893,Z 469.687,A -85,B 0,C 180,E1 -23049.412,E2 -23049.412} C_VEL
LIN {X 0,Y 171.822,Z 469.695,A -85,B 0,C 180,E1 -23050.557,E2 -23050.557} C_VEL
LIN {X 0,Y 172.503,Z 472.13,A -85,B 0,C 180,E1 -23051.505,E2 -23051.505} C_VEL
LIN {X 0,Y 174.232,Z 474.367,A -85,B 0,C 180,E1 -23053.262,E2 -23053.262} C_VEL
LIN {X 0,Y 176.539,Z 475.768,A -85,B 0,C 180,E1 -23055.218,E2 -23055.218} C_VEL
LIN {X 0,Y 178.14,Z 478.752,A -85,B 0,C 180,E1 -23056.693,E2 -23056.693} C_VEL
LIN {X 0,Y 180.959,Z 481.342,A -85,B 0,C 180,E1 -23058.832,E2 -23058.832} C_VEL
LIN {X 0,Y 183.232,Z 484.822,A -85,B 0,C 180,E1 -23060.523,E2 -23060.523} C_VEL
LIN {X 0,Y 185.265,Z 486.833,A -85,B 0,C 180,E1 -23061.844,E2 -23061.844} C_VEL
LIN {X 0,Y 187.863,Z 490.407,A -85,B 0,C 180,E1 -23063.515,E2 -23063.515} C_VEL
LIN {X 0,Y 189.299,Z 492.073,A -85,B 0,C 180,E1 -23064.374,E2 -23064.374} C_VEL
LIN {X 0,Y 193.494,Z 497.809,A -85,B 0,C 180,E1 -23066.768,E2 -23066.768} C_VEL
LIN {X 0,Y 196.602,Z 502.076,A -85,B 0,C 180,E1 -23068.389,E2 -23068.389} C_VEL
LIN {X 0,Y 200.681,Z 507.982,A -85,B 0,C 180,E1 -23070.403,E2 -23070.403} C_VEL
LIN {X 0,Y 207.826,Z 521.154,A -85,B 0,C 180,E1 -23073.733,E2 -23073.733} C_VEL
LIN {X 0,Y 213.444,Z 532.482,A -85,B 0,C 180,E1 -23076.128,E2 -23076.128} C_VEL
LIN {X 0,Y 219.886,Z 547.17,A -85,B 0,C 180,E1 -23078.711,E2 -23078.711} C_VEL
LIN {X 0,Y 221.825,Z 552.134,A -85,B 0,C 180,E1 -23079.466,E2 -23079.466} C_VEL
LIN {X 0,Y 218.743,Z 596.569,A -85,B 0,C 180,E1 -23080.779,E2 -23080.779} C_VEL
LIN {X 0,Y 217.814,Z 602.413,A -85,B 0,C 180,E1 -23080.817,E2 -23080.817} C_VEL
LIN {X 0,Y 212.253,Z 621.368,A -85,B 0,C 180,E1 -23080.289,E2 -23080.289} C_VEL
LIN {X 0,Y 211.374,Z 627.188,A -85,B 0,C 180,E1 -23080.381,E2 -23080.381} C_VEL
LIN {X 0,Y 209.458,Z 642.878,A -85,B 0,C 180,E1 -23081.07,E2 -23081.07} C_VEL
LIN {X 0,Y 206.754,Z 657.231,A -85,B 0,C 180,E1 -23081.962,E2 -23081.962} C_VEL
LIN {X 0,Y 203.173,Z 672.005,A -85,B 0,C 180,E1 -23083.232,E2 -23083.232} C_VEL
LIN {X 0,Y 199.256,Z 685.478,A -85,B 0,C 180,E1 -23084.778,E2 -23084.778} C_VEL
LIN {X 0,Y 194.776,Z 698.653,A -85,B 0,C 180,E1 -23086.719,E2 -23086.719} C_VEL
LIN {X 0,Y 189.995,Z 710.791,A -85,B 0,C 180,E1 -23088.96,E2 -23088.96} C_VEL
LIN {X 0,Y 185.606,Z 721.108,A -85,B 0,C 180,E1 -23091.333,E2 -23091.333} C_VEL
LIN {X 0,Y 180.7,Z 731.556,A -85,B 0,C 180,E1 -23094.309,E2 -23094.309} C_VEL
LIN {X 0,Y 176.466,Z 740.42,A -85,B 0,C 180,E1 -23097.475,E2 -23097.475} C_VEL
LIN {X 0,Y 172.689,Z 747.998,A -85,B 0,C 180,E1 -23100.765,E2 -23100.765} C_VEL
LIN {X 0,Y 169.454,Z 754.46,A -85,B 0,C 180,E1 -23104.183,E2 -23104.183} C_VEL
LIN {X 0,Y 166.103,Z 761.365,A -85,B 0,C 180,E1 -23108.783,E2 -23108.783} C_VEL
LIN {X 0,Y 163.731,Z 767.081,A -85,B 0,C 180,E1 -23113.798,E2 -23113.798} C_VEL
LIN {X 0,Y 162.587,Z 770.32,A -85,B 0,C 180,E1 -23117.517,E2 -23117.517} C_VEL
LIN {X 0,Y 161.87,Z 773.526,A -85,B 0,C 180,E1 -23122.515,E2 -23122.515} C_VEL
LIN {X 0,Y 161.763,Z 775.542,A -85,B 0,C 180,E1 -23127.792,E2 -23127.792} C_VEL
LIN {X 0,Y 161.906,Z 775.964,A -85,B 0,C 180,E1 -23129.999,E2 -23129.999} C_VEL
LIN {X 0,Y 161.742,Z 776.086,A -85,B 0,C 180,E1 -23134.984,E2 -23134.984} C_VEL
LIN {X 0,Y 162.119,Z 775.078,A -85,B 0,C 180,E1 -23139.984,E2 -23139.984} C_VEL
LIN {X 0,Y 163.291,Z 772.942,A -85,B 0,C 180,E1 -23144.964,E2 -23144.964} C_VEL
LIN {X 0,Y 165.563,Z 769.623,A -85,B 0,C 180,E1 -23149.85,E2 -23149.85} C_VEL
LIN {X 0,Y 168.865,Z 765.047,A -85,B 0,C 180,E1 -23154.593,E2 -23154.593} C_VEL
LIN {X 0,Y 173.233,Z 759.141,A -85,B 0,C 180,E1 -23159.131,E2 -23159.131} C_VEL
LIN {X 0,Y 178.767,Z 751.752,A -85,B 0,C 180,E1 -23163.392,E2 -23163.392} C_VEL
LIN {X 0,Y 184.223,Z 743.799,A -85,B 0,C 180,E1 -23166.988,E2 -23166.988} C_VEL
LIN {X 0,Y 190.338,Z 734.552,A -85,B 0,C 180,E1 -23170.251,E2 -23170.251} C_VEL
LIN {X 0,Y 196.224,Z 725.077,A -85,B 0,C 180,E1 -23172.881,E2 -23172.881} C_VEL
LIN {X 0,Y 202.428,Z 713.897,A -85,B 0,C 180,E1 -23175.374,E2 -23175.374} C_VEL
LIN {X 0,Y 208.535,Z 701.569,A -85,B 0,C 180,E1 -23177.523,E2 -23177.523} C_VEL
LIN {X 0,Y 214.247,Z 688.249,A -85,B 0,C 180,E1 -23179.336,E2 -23179.336} C_VEL
LIN {X 0,Y 219.019,Z 675.177,A -85,B 0,C 180,E1 -23180.724,E2 -23180.724} C_VEL
LIN {X 0,Y 223.379,Z 660.918,A -85,B 0,C 180,E1 -23181.862,E2 -23181.862} C_VEL
LIN {X 0,Y 227.067,Z 645.541,A -85,B 0,C 180,E1 -23182.75,E2 -23182.75} C_VEL
LIN {X 0,Y 229.655,Z 629.693,A -85,B 0,C 180,E1 -23183.41,E2 -23183.41} C_VEL
LIN {X 0,Y 235.694,Z 563.539,A -85,B 0,C 180,E1 -23185.2,E2 -23185.2} C_VEL
LIN {X 0,Y 232.549,Z 555.172,A -85,B 0,C 180,E1 -23187.285,E2 -23187.285} C_VEL
LIN {X 0,Y 229.257,Z 547.413,A -85,B 0,C 180,E1 -23189.686,E2 -23189.686} C_VEL
LIN {X 0,Y 226.487,Z 541.321,A -85,B 0,C 180,E1 -23191.987,E2 -23191.987} C_VEL
LIN {X 0,Y 224.328,Z 537.048,A -85,B 0,C 180,E1 -23193.985,E2 -23193.985} C_VEL
LIN {X 0,Y 222.744,Z 533.884,A -85,B 0,C 180,E1 -23195.697,E2 -23195.697} C_VEL
LIN {X 0,Y 220.307,Z 530.009,A -85,B 0,C 180,E1 -23198.724,E2 -23198.724} C_VEL
LIN {X 0,Y 218.246,Z 527.041,A -85,B 0,C 180,E1 -23202.239,E2 -23202.239} C_VEL
LIN {X 0,Y 217.675,Z 525.486,A -85,B 0,C 180,E1 -23203.848,E2 -23203.848} C_VEL
LIN {X 0,Y 216.726,Z 524.723,A -85,B 0,C 180,E1 -23210.669,E2 -23210.669} C_VEL
LIN {X 0,Y 218.204,Z 525.685,A -85,B 0,C 180,E1 -23215.795,E2 -23215.795} C_VEL
LIN {X 0,Y 220.197,Z 529.392,A -85,B 0,C 180,E1 -23219.504,E2 -23219.504} C_VEL
LIN {X 0,Y 220.926,Z 530.595,A -85,B 0,C 180,E1 -23220.543,E2 -23220.543} C_VEL
LIN {X 0,Y 223.438,Z 534.677,A -85,B 0,C 180,E1 -23223.469,E2 -23223.469} C_VEL
LIN {X 0,Y 225.952,Z 539.034,A -85,B 0,C 180,E1 -23225.884,E2 -23225.884} C_VEL
LIN {X 0,Y 229.039,Z 544.235,A -85,B 0,C 180,E1 -23228.384,E2 -23228.384} C_VEL
LIN {X 0,Y 233.031,Z 551.926,A -85,B 0,C 180,E1 -23231.18,E2 -23231.18} C_VEL
LIN {X 0,Y 235.987,Z 557.814,A -85,B 0,C 180,E1 -23233.01,E2 -23233.01} C_VEL
LIN {X 0,Y 234.546,Z 574.815,A -85,B 0,C 180,E1 -23233.499,E2 -23233.499} C_VEL
LIN {X 0,Y 230.136,Z 623.049,A -85,B 0,C 180,E1 -23234.827,E2 -23234.827} C_VEL
LIN {X 0,Y 227.664,Z 638.572,A -85,B 0,C 180,E1 -23235.486,E2 -23235.486} C_VEL
LIN {X 0,Y 224.521,Z 652.684,A -85,B 0,C 180,E1 -23236.363,E2 -23236.363} C_VEL
LIN {X 0,Y 220.259,Z 667.472,A -85,B 0,C 180,E1 -23237.596,E2 -23237.596} C_VEL
LIN {X 0,Y 215.021,Z 682.172,A -85,B 0,C 180,E1 -23239.23,E2 -23239.23} C_VEL
LIN {X 0,Y 209.457,Z 695.24,A -85,B 0,C 180,E1 -23241.095,E2 -23241.095} C_VEL
LIN {X 0,Y 203.624,Z 707.065,A -85,B 0,C 180,E1 -23243.231,E2 -23243.231} C_VEL
LIN {X 0,Y 197.016,Z 718.89,A -85,B 0,C 180,E1 -23245.961,E2 -23245.961} C_VEL
LIN {X 0,Y 190.651,Z 729.084,A -85,B 0,C 180,E1 -23248.972,E2 -23248.972} C_VEL
LIN {X 0,Y 184.957,Z 737.471,A -85,B 0,C 180,E1 -23252.14,E2 -23252.14} C_VEL
LIN {X 0,Y 178.933,Z 745.702,A -85,B 0,C 180,E1 -23256.098,E2 -23256.098} C_VEL
LIN {X 0,Y 173.783,Z 752.372,A -85,B 0,C 180,E1 -23260.321,E2 -23260.321} C_VEL
LIN {X 0,Y 169.276,Z 757.994,A -85,B 0,C 180,E1 -23265.108,E2 -23265.108} C_VEL
LIN {X 0,Y 165.657,Z 762.421,A -85,B 0,C 180,E1 -23270.48,E2 -23270.48} C_VEL
LIN {X 0,Y 163.249,Z 765.283,A -85,B 0,C 180,E1 -23275.97,E2 -23275.97} C_VEL
LIN {X 0,Y 161.863,Z 766.691,A -85,B 0,C 180,E1 -23281.472,E2 -23281.472} C_VEL
LIN {X 0,Y 161.356,Z 766.721,A -85,B 0,C 180,E1 -23286.923,E2 -23286.923} C_VEL
LIN {X 0,Y 161.51,Z 765.446,A -85,B 0,C 180,E1 -23292.268,E2 -23292.268} C_VEL
LIN {X 0,Y 162.336,Z 762.897,A -85,B 0,C 180,E1 -23297.5,E2 -23297.5} C_VEL
LIN {X 0,Y 163.926,Z 759.056,A -85,B 0,C 180,E1 -23302.612,E2 -23302.612} C_VEL
LIN {X 0,Y 166.308,Z 753.867,A -85,B 0,C 180,E1 -23307.579,E2 -23307.579} C_VEL
LIN {X 0,Y 169.668,Z 747.189,A -85,B 0,C 180,E1 -23312.375,E2 -23312.375} C_VEL
LIN {X 0,Y 173.311,Z 739.988,A -85,B 0,C 180,E1 -23316.404,E2 -23316.404} C_VEL
LIN {X 0,Y 177.743,Z 731.288,A -85,B 0,C 180,E1 -23320.25,E2 -23320.25} C_VEL
LIN {X 0,Y 182.819,Z 720.811,A -85,B 0,C 180,E1 -23323.903,E2 -23323.903} C_VEL
LIN {X 0,Y 188.116,Z 709.07,A -85,B 0,C 180,E1 -23327.111,E2 -23327.111} C_VEL
LIN {X 0,Y 193.111,Z 696.901,A -85,B 0,C 180,E1 -23329.729,E2 -23329.729} C_VEL
LIN {X 0,Y 197.848,Z 683.815,A -85,B 0,C 180,E1 -23331.957,E2 -23331.957} C_VEL
LIN {X 0,Y 202.147,Z 669.776,A -85,B 0,C 180,E1 -23333.84,E2 -23333.84} C_VEL
LIN {X 0,Y 205.733,Z 655.771,A -85,B 0,C 180,E1 -23335.279,E2 -23335.279} C_VEL
LIN {X 0,Y 208.658,Z 640.977,A -85,B 0,C 180,E1 -23336.439,E2 -23336.439} C_VEL
LIN {X 0,Y 210.96,Z 625.635,A -85,B 0,C 180,E1 -23337.264,E2 -23337.264} C_VEL
LIN {X 0,Y 212.617,Z 607.448,A -85,B 0,C 180,E1 -23337.886,E2 -23337.886} C_VEL
LIN {X 0,Y 217.057,Z 547.14,A -85,B 0,C 180,E1 -23339.662,E2 -23339.662} C_VEL
LIN {X 0,Y 210.195,Z 534.245,A -85,B 0,C 180,E1 -23342.361,E2 -23342.361} C_VEL
LIN {X 0,Y 203.999,Z 523.606,A -85,B 0,C 180,E1 -23345.025,E2 -23345.025} C_VEL
LIN {X 0,Y 197.302,Z 513.122,A -85,B 0,C 180,E1 -23348.183,E2 -23348.183} C_VEL
LIN {X 0,Y 191.552,Z 504.886,A -85,B 0,C 180,E1 -23351.197,E2 -23351.197} C_VEL
LIN {X 0,Y 188.496,Z 500.752,A -85,B 0,C 180,E1 -23352.953,E2 -23352.953} C_VEL
LIN {X 0,Y 185.734,Z 496.994,A -85,B 0,C 180,E1 -23354.659,E2 -23354.659} C_VEL
LIN {X 0,Y 182.821,Z 493.14,A -85,B 0,C 180,E1 -23356.583,E2 -23356.583} C_VEL
LIN {X 0,Y 179.442,Z 489.106,A -85,B 0,C 180,E1 -23359.016,E2 -23359.016} C_VEL
LIN {X 0,Y 178.321,Z 487.454,A -85,B 0,C 180,E1 -23359.903,E2 -23359.903} C_VEL
LIN {X 0,Y 175.601,Z 484.702,A -85,B 0,C 180,E1 -23362.101,E2 -23362.101} C_VEL
LIN {X 0,Y 174.16,Z 482.222,A -85,B 0,C 180,E1 -23363.49,E2 -23363.49} C_VEL
LIN {X 0,Y 171.535,Z 480.236,A -85,B 0,C 180,E1 -23365.946,E2 -23365.946} C_VEL
LIN {X 0,Y 169.844,Z 477.275,A -85,B 0,C 180,E1 -23367.957,E2 -23367.957} C_VEL
LIN {X 0,Y 169.519,Z 476.585,A -85,B 0,C 180,E1 -23368.388,E2 -23368.388} C_VEL
LIN {X 0,Y 166.239,Z 474.617,A -85,B 0,C 180,E1 -23372.529,E2 -23372.529} C_VEL
LIN {X 0,Y 164.713,Z 471.997,A -85,B 0,C 180,E1 -23375.332,E2 -23375.332} C_VEL
LIN {X 0,Y 164.381,Z 470.607,A -85,B 0,C 180,E1 -23376.203,E2 -23376.203} C_VEL
LIN {X 0,Y 164.488,Z 470.621,A -85,B 0,C 180,E1 -23380.051,E2 -23380.051} C_VEL
LIN {X 0,Y 164.539,Z 470.594,A -85,B 0,C 180,E1 -23385.15,E2 -23385.15} C_VEL
LIN {X 0,Y 164.808,Z 470.551,A -85,B 0,C 180,E1 -23390.178,E2 -23390.178} C_VEL
LIN {X 0,Y 164.857,Z 470.562,A -85,B 0,C 180,E1 -23392.652,E2 -23392.652} C_VEL
LIN {X 0,Y 165.052,Z 470.522,A -85,B 0,C 180,E1 -23397.559,E2 -23397.559} C_VEL
LIN {X 0,Y 165.298,Z 470.517,A -85,B 0,C 180,E1 -23399.999,E2 -23399.999} C_VEL
LIN {X 0,Y 165.029,Z 470.577,A -85,B 0,C 180,E1 -23402.516,E2 -23402.516} C_VEL
LIN {X 0,Y 165.521,Z 472.774,A -85,B 0,C 180,E1 -23403.727,E2 -23403.727} C_VEL
LIN {X 0,Y 166.972,Z 474.837,A -85,B 0,C 180,E1 -23406.04,E2 -23406.04} C_VEL
LIN {X 0,Y 170.051,Z 476.806,A -85,B 0,C 180,E1 -23409.777,E2 -23409.777} C_VEL
LIN {X 0,Y 171.388,Z 479.702,A -85,B 0,C 180,E1 -23411.448,E2 -23411.448} C_VEL
LIN {X 0,Y 173.752,Z 481.892,A -85,B 0,C 180,E1 -23413.731,E2 -23413.731} C_VEL
LIN {X 0,Y 174.697,Z 482.677,A -85,B 0,C 180,E1 -23414.562,E2 -23414.562} C_VEL
LIN {X 0,Y 176.644,Z 485.717,A -85,B 0,C 180,E1 -23416.337,E2 -23416.337} C_VEL
LIN {X 0,Y 178.906,Z 487.93,A -85,B 0,C 180,E1 -23418.122,E2 -23418.122} C_VEL
LIN {X 0,Y 181.413,Z 491.557,A -85,B 0,C 180,E1 -23420.034,E2 -23420.034} C_VEL
LIN {X 0,Y 183.023,Z 493.278,A -85,B 0,C 180,E1 -23421.127,E2 -23421.127} C_VEL
LIN {X 0,Y 186.031,Z 497.191,A -85,B 0,C 180,E1 -23423.09,E2 -23423.09} C_VEL
LIN {X 0,Y 190.626,Z 503.574,A -85,B 0,C 180,E1 -23425.866,E2 -23425.866} C_VEL
LIN {X 0,Y 195.698,Z 510.699,A -85,B 0,C 180,E1 -23428.583,E2 -23428.583} C_VEL
LIN {X 0,Y 199.464,Z 517.13,A -85,B 0,C 180,E1 -23430.508,E2 -23430.508} C_VEL
LIN {X 0,Y 206.036,Z 529.879,A -85,B 0,C 180,E1 -23433.625,E2 -23433.625} C_VEL
LIN {X 0,Y 211.693,Z 542.099,A -85,B 0,C 180,E1 -23436.106,E2 -23436.106} C_VEL
LIN {X 0,Y 216.771,Z 554.468,A -85,B 0,C 180,E1 -23438.213,E2 -23438.213} C_VEL
LIN {X 0,Y 211.374,Z 627.188,A -85,B 0,C 180,E1 -23440.381,E2 -23440.381} C_VEL
LIN {X 0,Y 210.817,Z 631.072,A -85,B 0,C 180,E1 -23440.463,E2 -23440.463} C_VEL
LIN {X 0,Y 209.213,Z 636.779,A -85,B 0,C 180,E1 -23440.465,E2 -23440.465} C_VEL
LIN {X 0,Y 203.235,Z 651.533,A -85,B 0,C 180,E1 -23440.328,E2 -23440.328} C_VEL
LIN {X 0,Y 202.038,Z 655.269,A -85,B 0,C 180,E1 -23440.468,E2 -23440.468} C_VEL
LIN {X 0,Y 201.597,Z 657.142,A -85,B 0,C 180,E1 -23440.602,E2 -23440.602} C_VEL
LIN {X 0,Y 197.773,Z 672.348,A -85,B 0,C 180,E1 -23441.923,E2 -23441.923} C_VEL
LIN {X 0,Y 193.325,Z 686.954,A -85,B 0,C 180,E1 -23443.651,E2 -23443.651} C_VEL
LIN {X 0,Y 188.564,Z 700.117,A -85,B 0,C 180,E1 -23445.665,E2 -23445.665} C_VEL
LIN {X 0,Y 183.656,Z 711.98,A -85,B 0,C 180,E1 -23447.957,E2 -23447.957} C_VEL
LIN {X 0,Y 179.153,Z 722.093,A -85,B 0,C 180,E1 -23450.395,E2 -23450.395} C_VEL
LIN {X 0,Y 174.116,Z 732.399,A -85,B 0,C 180,E1 -23453.461,E2 -23453.461} C_VEL
LIN {X 0,Y 169.735,Z 741.106,A -85,B 0,C 180,E1 -23456.726,E2 -23456.726} C_VEL
LIN {X 0,Y 165.833,Z 748.529,A -85,B 0,C 180,E1 -23460.133,E2 -23460.133} C_VEL
LIN {X 0,Y 161.985,Z 755.831,A -85,B 0,C 180,E1 -23464.285,E2 -23464.285} C_VEL
LIN {X 0,Y 158.621,Z 762.579,A -85,B 0,C 180,E1 -23469.239,E2 -23469.239} C_VEL
LIN {X 0,Y 156.349,Z 767.839,A -85,B 0,C 180,E1 -23474.352,E2 -23474.352} C_VEL
LIN {X 0,Y 155.1,Z 771.745,A -85,B 0,C 180,E1 -23479.556,E2 -23479.556} C_VEL
LIN {X 0,Y 154.674,Z 774.35,A -85,B 0,C 180,E1 -23484.785,E2 -23484.785} C_VEL
LIN {X 0,Y 154.804,Z 775.714,A -85,B 0,C 180,E1 -23489.999,E2 -23489.999} C_VEL
LIN {X 0,Y 154.646,Z 775.891,A -85,B 0,C 180,E1 -23495.213,E2 -23495.213} C_VEL
LIN {X 0,Y 155.102,Z 774.939,A -85,B 0,C 180,E1 -23500.441,E2 -23500.441} C_VEL
LIN {X 0,Y 156.39,Z 772.864,A -85,B 0,C 180,E1 -23505.641,E2 -23505.641} C_VEL
LIN {X 0,Y 158.848,Z 769.581,A -85,B 0,C 180,E1 -23510.727,E2 -23510.727} C_VEL
LIN {X 0,Y 162.392,Z 765.071,A -85,B 0,C 180,E1 -23515.642,E2 -23515.642} C_VEL
LIN {X 0,Y 167.007,Z 759.237,A -85,B 0,C 180,E1 -23520.328,E2 -23520.328} C_VEL
LIN {X 0,Y 172.863,Z 751.944,A -85,B 0,C 180,E1 -23524.692,E2 -23524.692} C_VEL
LIN {X 0,Y 178.418,Z 744.329,A -85,B 0,C 180,E1 -23528.272,E2 -23528.272} C_VEL
LIN {X 0,Y 184.987,Z 734.956,A -85,B 0,C 180,E1 -23531.669,E2 -23531.669} C_VEL
LIN {X 0,Y 191.108,Z 725.597,A -85,B 0,C 180,E1 -23534.322,E2 -23534.322} C_VEL
LIN {X 0,Y 198.08,Z 713.527,A -85,B 0,C 180,E1 -23537.034,E2 -23537.034} C_VEL
LIN {X 0,Y 204.829,Z 700.291,A -85,B 0,C 180,E1 -23539.314,E2 -23539.314} C_VEL
LIN {X 0,Y 210.349,Z 687.899,A -85,B 0,C 180,E1 -23540.967,E2 -23540.967} C_VEL
LIN {X 0,Y 215.288,Z 674.82,A -85,B 0,C 180,E1 -23542.336,E2 -23542.336} C_VEL
LIN {X 0,Y 219.8,Z 660.512,A -85,B 0,C 180,E1 -23543.45,E2 -23543.45} C_VEL
LIN {X 0,Y 223.569,Z 645.082,A -85,B 0,C 180,E1 -23544.33,E2 -23544.33} C_VEL
LIN {X 0,Y 226.252,Z 628.954,A -85,B 0,C 180,E1 -23544.981,E2 -23544.981} C_VEL
LIN {X 0,Y 232.102,Z 566.504,A -85,B 0,C 180,E1 -23546.678,E2 -23546.678} C_VEL
LIN {X 0,Y 229.055,Z 558.165,A -85,B 0,C 180,E1 -23548.923,E2 -23548.923} C_VEL
LIN {X 0,Y 225.452,Z 549.449,A -85,B 0,C 180,E1 -23551.916,E2 -23551.916} C_VEL
LIN {X 0,Y 222.781,Z 543.725,A -85,B 0,C 180,E1 -23554.498,E2 -23554.498} C_VEL
LIN {X 0,Y 221.231,Z 540.444,A -85,B 0,C 180,E1 -23556.266,E2 -23556.266} C_VEL
LIN {X 0,Y 218.925,Z 536.702,A -85,B 0,C 180,E1 -23559.322,E2 -23559.322} C_VEL
LIN {X 0,Y 217.023,Z 533.581,A -85,B 0,C 180,E1 -23562.941,E2 -23562.941} C_VEL
LIN {X 0,Y 216.607,Z 532.453,A -85,B 0,C 180,E1 -23564.212,E2 -23564.212} C_VEL
LIN {X 0,Y 215.8,Z 531.737,A -85,B 0,C 180,E1 -23570.629,E2 -23570.629} C_VEL
LIN {X 0,Y 217.146,Z 532.72,A -85,B 0,C 180,E1 -23575.538,E2 -23575.538} C_VEL
LIN {X 0,Y 219.002,Z 536.276,A -85,B 0,C 180,E1 -23579.167,E2 -23579.167} C_VEL
LIN {X 0,Y 221.682,Z 540.805,A -85,B 0,C 180,E1 -23582.661,E2 -23582.661} C_VEL
LIN {X 0,Y 224.69,Z 546.333,A -85,B 0,C 180,E1 -23585.71,E2 -23585.71} C_VEL
LIN {X 0,Y 227.176,Z 550.804,A -85,B 0,C 180,E1 -23587.804,E2 -23587.804} C_VEL
LIN {X 0,Y 230.679,Z 557.851,A -85,B 0,C 180,E1 -23590.401,E2 -23590.401} C_VEL
LIN {X 0,Y 232.45,Z 561.463,A -85,B 0,C 180,E1 -23591.589,E2 -23591.589} C_VEL
LIN {X 0,Y 226.688,Z 622.911,A -85,B 0,C 180,E1 -23593.27,E2 -23593.27} C_VEL
LIN {X 0,Y 224.124,Z 638.606,A -85,B 0,C 180,E1 -23593.918,E2 -23593.918} C_VEL
LIN {X 0,Y 220.811,Z 653.055,A -85,B 0,C 180,E1 -23594.806,E2 -23594.806} C_VEL
LIN {X 0,Y 216.579,Z 667.343,A -85,B 0,C 180,E1 -23595.992,E2 -23595.992} C_VEL
LIN {X 0,Y 211.895,Z 680.188,A -85,B 0,C 180,E1 -23597.368,E2 -23597.368} C_VEL
LIN {X 0,Y 206.389,Z 692.968,A -85,B 0,C 180,E1 -23599.107,E2 -23599.107} C_VEL
LIN {X 0,Y 200.566,Z 704.609,A -85,B 0,C 180,E1 -23601.104,E2 -23601.104} C_VEL
LIN {X 0,Y 194.172,Z 716.026,A -85,B 0,C 180,E1 -23603.618,E2 -23603.618} C_VEL
LIN {X 0,Y 188.053,Z 725.669,A -85,B 0,C 180,E1 -23606.246,E2 -23606.246} C_VEL
LIN {X 0,Y 181.657,Z 734.958,A -85,B 0,C 180,E1 -23609.491,E2 -23609.491} C_VEL
LIN {X 0,Y 175.855,Z 742.725,A -85,B 0,C 180,E1 -23612.941,E2 -23612.941} C_VEL
LIN {X 0,Y 170.622,Z 749.128,A -85,B 0,C 180,E1 -23616.565,E2 -23616.565} C_VEL
LIN {X 0,Y 166.187,Z 754.435,A -85,B 0,C 180,E1 -23620.432,E2 -23620.432} C_VEL
LIN {X 0,Y 162.292,Z 758.963,A -85,B 0,C 180,E1 -23624.686,E2 -23624.686} C_VEL
LIN {X 0,Y 159.494,Z 762.065,A -85,B 0,C 180,E1 -23628.629,E2 -23628.629} C_VEL
LIN {X 0,Y 156.706,Z 765.146,A -85,B 0,C 180,E1 -23634.338,E2 -23634.338} C_VEL
LIN {X 0,Y 155.014,Z 766.76,A -85,B 0,C 180,E1 -23640.087,E2 -23640.087} C_VEL
LIN {X 0,Y 154.298,Z 766.993,A -85,B 0,C 180,E1 -23645.801,E2 -23645.801} C_VEL
LIN {X 0,Y 154.321,Z 765.915,A -85,B 0,C 180,E1 -23651.412,E2 -23651.412} C_VEL
LIN {X 0,Y 155.076,Z 763.563,A -85,B 0,C 180,E1 -23656.905,E2 -23656.905} C_VEL
LIN {X 0,Y 156.649,Z 759.92,A -85,B 0,C 180,E1 -23662.266,E2 -23662.266} C_VEL
LIN {X 0,Y 159.01,Z 754.943,A -85,B 0,C 180,E1 -23667.468,E2 -23667.468} C_VEL
LIN {X 0,Y 162.385,Z 748.496,A -85,B 0,C 180,E1 -23672.482,E2 -23672.482} C_VEL
LIN {X 0,Y 166.721,Z 740.396,A -85,B 0,C 180,E1 -23677.266,E2 -23677.266} C_VEL
LIN {X 0,Y 171.353,Z 731.735,A -85,B 0,C 180,E1 -23681.235,E2 -23681.235} C_VEL
LIN {X 0,Y 176.616,Z 721.306,A -85,B 0,C 180,E1 -23684.991,E2 -23684.991} C_VEL
LIN {X 0,Y 181.662,Z 710.611,A -85,B 0,C 180,E1 -23688.03,E2 -23688.03} C_VEL
LIN {X 0,Y 186.722,Z 698.932,A -85,B 0,C 180,E1 -23690.664,E2 -23690.664} C_VEL
LIN {X 0,Y 191.416,Z 686.751,A -85,B 0,C 180,E1 -23692.858,E2 -23692.858} C_VEL
LIN {X 0,Y 195.648,Z 674.055,A -85,B 0,C 180,E1 -23694.683,E2 -23694.683} C_VEL
LIN {X 0,Y 199.533,Z 660.042,A -85,B 0,C 180,E1 -23696.263,E2 -23696.263} C_VEL
LIN {X 0,Y 202.805,Z 645.648,A -85,B 0,C 180,E1 -23697.474,E2 -23697.474} C_VEL
LIN {X 0,Y 205.369,Z 630.343,A -85,B 0,C 180,E1 -23698.418,E2 -23698.418} C_VEL
LIN {X 0,Y 207.073,Z 614.988,A -85,B 0,C 180,E1 -23699.033,E2 -23699.033} C_VEL
LIN {X 0,Y 211.999,Z 549.901,A -85,B 0,C 180,E1 -23700.978,E2 -23700.978} C_VEL
LIN {X 0,Y 205.375,Z 537.293,A -85,B 0,C 180,E1 -23703.763,E2 -23703.763} C_VEL
LIN {X 0,Y 200.035,Z 528.041,A -85,B 0,C 180,E1 -23706.186,E2 -23706.186} C_VEL
LIN {X 0,Y 193.811,Z 518.149,A -85,B 0,C 180,E1 -23709.294,E2 -23709.294} C_VEL
LIN {X 0,Y 188.18,Z 509.925,A -85,B 0,C 180,E1 -23712.417,E2 -23712.417} C_VEL
LIN {X 0,Y 183.183,Z 503.023,A -85,B 0,C 180,E1 -23715.545,E2 -23715.545} C_VEL
LIN {X 0,Y 179.782,Z 498.561,A -85,B 0,C 180,E1 -23717.922,E2 -23717.922} C_VEL
LIN {X 0,Y 176.962,Z 494.854,A -85,B 0,C 180,E1 -23720.095,E2 -23720.095} C_VEL
LIN {X 0,Y 175.989,Z 493.699,A -85,B 0,C 180,E1 -23720.884,E2 -23720.884} C_VEL
LIN {X 0,Y 173.265,Z 490.48,A -85,B 0,C 180,E1 -23723.27,E2 -23723.27} C_VEL
LIN {X 0,Y 172.246,Z 488.827,A -85,B 0,C 180,E1 -23724.296,E2 -23724.296} C_VEL
LIN {X 0,Y 169.693,Z 486.597,A -85,B 0,C 180,E1 -23726.835,E2 -23726.835} C_VEL
LIN {X 0,Y 167.949,Z 483.41,A -85,B 0,C 180,E1 -23729.061,E2 -23729.061} C_VEL
LIN {X 0,Y 164.83,Z 481.306,A -85,B 0,C 180,E1 -23733.229,E2 -23733.229} C_VEL
LIN {X 0,Y 163.29,Z 478.393,A -85,B 0,C 180,E1 -23736.286,E2 -23736.286} C_VEL
LIN {X 0,Y 163.09,Z 477.571,A -85,B 0,C 180,E1 -23736.844,E2 -23736.844} C_VEL
LIN {X 0,Y 160.197,Z 476.155,A -85,B 0,C 180,E1 -23747.328,E2 -23747.328} C_VEL
LIN {X 0,Y 160.437,Z 476.13,A -85,B 0,C 180,E1 -23752.448,E2 -23752.448} C_VEL
LIN {X 0,Y 163.645,Z 477.608,A -85,B 0,C 180,E1 -23761.768,E2 -23761.768} C_VEL
LIN {X 0,Y 164.491,Z 480.176,A -85,B 0,C 180,E1 -23763.674,E2 -23763.674} C_VEL
LIN {X 0,Y 166.699,Z 482.492,A -85,B 0,C 180,E1 -23766.961,E2 -23766.961} C_VEL
LIN {X 0,Y 168.433,Z 483.647,A -85,B 0,C 180,E1 -23769.077,E2 -23769.077} C_VEL
LIN {X 0,Y 169.948,Z 486.589,A -85,B 0,C 180,E1 -23770.996,E2 -23770.996} C_VEL
LIN {X 0,Y 172.814,Z 489.215,A -85,B 0,C 180,E1 -23773.807,E2 -23773.807} C_VEL
LIN {X 0,Y 175.057,Z 492.54,A -85,B 0,C 180,E1 -23775.9,E2 -23775.9} C_VEL
LIN {X 0,Y 176.892,Z 494.524,A -85,B 0,C 180,E1 -23777.403,E2 -23777.403} C_VEL
LIN {X 0,Y 179.714,Z 498.371,A -85,B 0,C 180,E1 -23779.609,E2 -23779.609} C_VEL
LIN {X 0,Y 181.222,Z 500.326,A -85,B 0,C 180,E1 -23780.69,E2 -23780.69} C_VEL
LIN {X 0,Y 184.913,Z 505.285,A -85,B 0,C 180,E1 -23783.148,E2 -23783.148} C_VEL
LIN {X 0,Y 188.184,Z 509.883,A -85,B 0,C 180,E1 -23785.167,E2 -23785.167} C_VEL
LIN {X 0,Y 193.494,Z 517.615,A -85,B 0,C 180,E1 -23788.121,E2 -23788.121} C_VEL
LIN {X 0,Y 198.668,Z 527.417,A -85,B 0,C 180,E1 -23790.846,E2 -23790.846} C_VEL
LIN {X 0,Y 204.963,Z 540.399,A -85,B 0,C 180,E1 -23793.862,E2 -23793.862} C_VEL
LIN {X 0,Y 211.014,Z 554.874,A -85,B 0,C 180,E1 -23796.574,E2 -23796.574} C_VEL
LIN {X 0,Y 211.79,Z 556.801,A -85,B 0,C 180,E1 -23796.904,E2 -23796.904} C_VEL
LIN {X 0,Y 206.077,Z 630.221,A -85,B 0,C 180,E1 -23799.116,E2 -23799.116} C_VEL
LIN {X 0,Y 203.791,Z 646.307,A -85,B 0,C 180,E1 -23799.885,E2 -23799.885} C_VEL
LIN {X 0,Y 201.597,Z 657.142,A -85,B 0,C 180,E1 -23800.602,E2 -23800.602} C_VEL
LIN {X 0,Y 199.84,Z 662.741,A -85,B 0,C 180,E1 -23800.912,E2 -23800.912} C_VEL
LIN {X 0,Y 195.395,Z 671.534,A -85,B 0,C 180,E1 -23801.146,E2 -23801.146} C_VEL
LIN {X 0,Y 190.661,Z 680.178,A -85,B 0,C 180,E1 -23801.514,E2 -23801.514} C_VEL
LIN {X 0,Y 188.47,Z 685.349,A -85,B 0,C 180,E1 -23802.046,E2 -23802.046} C_VEL
LIN {X 0,Y 183.51,Z 698.89,A -85,B 0,C 180,E1 -23804.103,E2 -23804.103} C_VEL
LIN {X 0,Y 178.418,Z 710.93,A -85,B 0,C 180,E1 -23806.421,E2 -23806.421} C_VEL
LIN {X 0,Y 172.754,Z 722.992,A -85,B 0,C 180,E1 -23809.388,E2 -23809.388} C_VEL
LIN {X 0,Y 167.558,Z 733.124,A -85,B 0,C 180,E1 -23812.542,E2 -23812.542} C_VEL
LIN {X 0,Y 163.033,Z 741.751,A -85,B 0,C 180,E1 -23815.915,E2 -23815.915} C_VEL
LIN {X 0,Y 158.352,Z 750.167,A -85,B 0,C 180,E1 -23820.045,E2 -23820.045} C_VEL
LIN {X 0,Y 154.517,Z 757.125,A -85,B 0,C 180,E1 -23824.398,E2 -23824.398} C_VEL
LIN {X 0,Y 151.209,Z 763.558,A -85,B 0,C 180,E1 -23829.598,E2 -23829.598} C_VEL
LIN {X 0,Y 148.996,Z 768.519,A -85,B 0,C 180,E1 -23834.962,E2 -23834.962} C_VEL
LIN {X 0,Y 148.069,Z 771.396,A -85,B 0,C 180,E1 -23839.054,E2 -23839.054} C_VEL
LIN {X 0,Y 147.599,Z 774.04,A -85,B 0,C 180,E1 -23844.534,E2 -23844.534} C_VEL
LIN {X 0,Y 147.715,Z 775.463,A -85,B 0,C 180,E1 -23849.998,E2 -23849.998} C_VEL
LIN {X 0,Y 147.551,Z 775.696,A -85,B 0,C 180,E1 -23855.465,E2 -23855.465} C_VEL
LIN {X 0,Y 148.073,Z 774.806,A -85,B 0,C 180,E1 -23860.942,E2 -23860.942} C_VEL
LIN {X 0,Y 149.518,Z 772.772,A -85,B 0,C 180,E1 -23866.379,E2 -23866.379} C_VEL
LIN {X 0,Y 152.175,Z 769.54,A -85,B 0,C 180,E1 -23871.681,E2 -23871.681} C_VEL
LIN {X 0,Y 155.953,Z 765.108,A -85,B 0,C 180,E1 -23876.783,E2 -23876.783} C_VEL
LIN {X 0,Y 160.868,Z 759.365,A -85,B 0,C 180,E1 -23881.616,E2 -23881.616} C_VEL
LIN {X 0,Y 167.053,Z 752.154,A -85,B 0,C 180,E1 -23886.083,E2 -23886.083} C_VEL
LIN {X 0,Y 172.885,Z 744.631,A -85,B 0,C 180,E1 -23889.733,E2 -23889.733} C_VEL
LIN {X 0,Y 179.76,Z 735.379,A -85,B 0,C 180,E1 -23893.17,E2 -23893.17} C_VEL
LIN {X 0,Y 186.122,Z 726.126,A -85,B 0,C 180,E1 -23895.841,E2 -23895.841} C_VEL
LIN {X 0,Y 192.778,Z 715.221,A -85,B 0,C 180,E1 -23898.359,E2 -23898.359} C_VEL
LIN {X 0,Y 199.309,Z 703.261,A -85,B 0,C 180,E1 -23900.504,E2 -23900.504} C_VEL
LIN {X 0,Y 205.371,Z 690.423,A -85,B 0,C 180,E1 -23902.31,E2 -23902.31} C_VEL
LIN {X 0,Y 210.439,Z 677.919,A -85,B 0,C 180,E1 -23903.675,E2 -23903.675} C_VEL
LIN {X 0,Y 215.023,Z 664.553,A -85,B 0,C 180,E1 -23904.795,E2 -23904.795} C_VEL
LIN {X 0,Y 219.048,Z 649.887,A -85,B 0,C 180,E1 -23905.705,E2 -23905.705} C_VEL
LIN {X 0,Y 222.108,Z 634.43,A -85,B 0,C 180,E1 -23906.403,E2 -23906.403} C_VEL
LIN {X 0,Y 224.268,Z 616.789,A -85,B 0,C 180,E1 -23906.931,E2 -23906.931} C_VEL
LIN {X 0,Y 228.726,Z 569.628,A -85,B 0,C 180,E1 -23908.196,E2 -23908.196} C_VEL
LIN {X 0,Y 225.567,Z 560.843,A -85,B 0,C 180,E1 -23910.779,E2 -23910.779} C_VEL
LIN {X 0,Y 222.662,Z 553.618,A -85,B 0,C 180,E1 -23913.5,E2 -23913.5} C_VEL
LIN {X 0,Y 219.932,Z 547.346,A -85,B 0,C 180,E1 -23916.608,E2 -23916.608} C_VEL
LIN {X 0,Y 217.718,Z 543.551,A -85,B 0,C 180,E1 -23919.692,E2 -23919.692} C_VEL
LIN {X 0,Y 215.914,Z 540.396,A -85,B 0,C 180,E1 -23923.377,E2 -23923.377} C_VEL
LIN {X 0,Y 215.699,Z 539.531,A -85,B 0,C 180,E1 -23924.143,E2 -23924.143} C_VEL
LIN {X 0,Y 214.868,Z 538.779,A -85,B 0,C 180,E1 -23930.588,E2 -23930.588} C_VEL
LIN {X 0,Y 216.087,Z 539.715,A -85,B 0,C 180,E1 -23935.265,E2 -23935.265} C_VEL
LIN {X 0,Y 218.289,Z 544.063,A -85,B 0,C 180,E1 -23939.583,E2 -23939.583} C_VEL
LIN {X 0,Y 220.332,Z 547.774,A -85,B 0,C 180,E1 -23942.294,E2 -23942.294} C_VEL
LIN {X 0,Y 223.303,Z 553.392,A -85,B 0,C 180,E1 -23945.418,E2 -23945.418} C_VEL
LIN {X 0,Y 225.814,Z 558.378,A -85,B 0,C 180,E1 -23947.617,E2 -23947.617} C_VEL
LIN {X 0,Y 229.032,Z 565.109,A -85,B 0,C 180,E1 -23950.077,E2 -23950.077} C_VEL
LIN {X 0,Y 223.365,Z 623.61,A -85,B 0,C 180,E1 -23951.687,E2 -23951.687} C_VEL
LIN {X 0,Y 220.588,Z 639.706,A -85,B 0,C 180,E1 -23952.358,E2 -23952.358} C_VEL
LIN {X 0,Y 217.437,Z 652.953,A -85,B 0,C 180,E1 -23953.169,E2 -23953.169} C_VEL
LIN {X 0,Y 213.069,Z 667.234,A -85,B 0,C 180,E1 -23954.329,E2 -23954.329} C_VEL
LIN {X 0,Y 207.623,Z 681.647,A -85,B 0,C 180,E1 -23955.866,E2 -23955.866} C_VEL
LIN {X 0,Y 201.86,Z 694.381,A -85,B 0,C 180,E1 -23957.624,E2 -23957.624} C_VEL
LIN {X 0,Y 195.176,Z 707.017,A -85,B 0,C 180,E1 -23959.845,E2 -23959.845} C_VEL
LIN {X 0,Y 188.273,Z 718.557,A -85,B 0,C 180,E1 -23962.503,E2 -23962.503} C_VEL
LIN {X 0,Y 181.045,Z 729.133,A -85,B 0,C 180,E1 -23965.608,E2 -23965.608} C_VEL
LIN {X 0,Y 174.665,Z 737.648,A -85,B 0,C 180,E1 -23968.872,E2 -23968.872} C_VEL
LIN {X 0,Y 167.905,Z 745.943,A -85,B 0,C 180,E1 -23972.967,E2 -23972.967} C_VEL
LIN {X 0,Y 162.006,Z 752.672,A -85,B 0,C 180,E1 -23977.398,E2 -23977.398} C_VEL
LIN {X 0,Y 157.072,Z 758.016,A -85,B 0,C 180,E1 -23982.157,E2 -23982.157} C_VEL
LIN {X 0,Y 153.126,Z 762.122,A -85,B 0,C 180,E1 -23987.253,E2 -23987.253} C_VEL
LIN {X 0,Y 150.204,Z 765.065,A -85,B 0,C 180,E1 -23992.696,E2 -23992.696} C_VEL
LIN {X 0,Y 148.255,Z 766.832,A -85,B 0,C 180,E1 -23998.572,E2 -23998.572} C_VEL
LIN {X 0,Y 147.264,Z 767.266,A -85,B 0,C 180,E1 -24004.565,E2 -24004.565} C_VEL
LIN {X 0,Y 147.156,Z 766.379,A -85,B 0,C 180,E1 -24010.471,E2 -24010.471} C_VEL
LIN {X 0,Y 147.452,Z 765.452,A -85,B 0,C 180,E1 -24013.384,E2 -24013.384} C_VEL
LIN {X 0,Y 148.476,Z 762.657,A -85,B 0,C 180,E1 -24019.088,E2 -24019.088} C_VEL
LIN {X 0,Y 150.418,Z 758.544,A -85,B 0,C 180,E1 -24024.64,E2 -24024.64} C_VEL
LIN {X 0,Y 153.278,Z 753.056,A -85,B 0,C 180,E1 -24030.001,E2 -24030.001} C_VEL
LIN {X 0,Y 157.217,Z 746.047,A -85,B 0,C 180,E1 -24035.131,E2 -24035.131} C_VEL
LIN {X 0,Y 161.418,Z 738.49,A -85,B 0,C 180,E1 -24039.398,E2 -24039.398} C_VEL
LIN {X 0,Y 166.403,Z 729.563,A -85,B 0,C 180,E1 -24043.346,E2 -24043.346} C_VEL
LIN {X 0,Y 171.346,Z 720.08,A -85,B 0,C 180,E1 -24046.686,E2 -24046.686} C_VEL
LIN {X 0,Y 176.673,Z 709.1,A -85,B 0,C 180,E1 -24049.764,E2 -24049.764} C_VEL
LIN {X 0,Y 181.987,Z 697.078,A -85,B 0,C 180,E1 -24052.419,E2 -24052.419} C_VEL
LIN {X 0,Y 187.076,Z 683.941,A -85,B 0,C 180,E1 -24054.706,E2 -24054.706} C_VEL
LIN {X 0,Y 191.262,Z 671.237,A -85,B 0,C 180,E1 -24056.459,E2 -24056.459} C_VEL
LIN {X 0,Y 195.344,Z 656.395,A -85,B 0,C 180,E1 -24058.032,E2 -24058.032} C_VEL
LIN {X 0,Y 198.467,Z 641.671,A -85,B 0,C 180,E1 -24059.211,E2 -24059.211} C_VEL
LIN {X 0,Y 201.052,Z 625.532,A -85,B 0,C 180,E1 -24060.08,E2 -24060.08} C_VEL
LIN {X 0,Y 203.08,Z 603.807,A -85,B 0,C 180,E1 -24060.807,E2 -24060.807} C_VEL
LIN {X 0,Y 207.094,Z 552.624,A -85,B 0,C 180,E1 -24062.341,E2 -24062.341} C_VEL
LIN {X 0,Y 199.889,Z 538.921,A -85,B 0,C 180,E1 -24065.579,E2 -24065.579} C_VEL
LIN {X 0,Y 193.527,Z 528.128,A -85,B 0,C 180,E1 -24068.749,E2 -24068.749} C_VEL
LIN {X 0,Y 186.896,Z 517.751,A -85,B 0,C 180,E1 -24072.457,E2 -24072.457} C_VEL
LIN {X 0,Y 180.931,Z 509.336,A -85,B 0,C 180,E1 -24076.282,E2 -24076.282} C_VEL
LIN {X 0,Y 177.4,Z 504.65,A -85,B 0,C 180,E1 -24078.869,E2 -24078.869} C_VEL
LIN {X 0,Y 174.215,Z 500.339,A -85,B 0,C 180,E1 -24081.471,E2 -24081.471} C_VEL
LIN {X 0,Y 171.367,Z 496.877,A -85,B 0,C 180,E1 -24084.084,E2 -24084.084} C_VEL
LIN {X 0,Y 170.556,Z 495.534,A -85,B 0,C 180,E1 -24084.924,E2 -24084.924} C_VEL
LIN {X 0,Y 167.945,Z 493.002,A -85,B 0,C 180,E1 -24087.677,E2 -24087.677} C_VEL
LIN {X 0,Y 166.292,Z 490.173,A -85,B 0,C 180,E1 -24089.875,E2 -24089.875} C_VEL
LIN {X 0,Y 163.454,Z 488.016,A -85,B 0,C 180,E1 -24093.914,E2 -24093.914} C_VEL
LIN {X 0,Y 161.911,Z 484.789,A -85,B 0,C 180,E1 -24097.257,E2 -24097.257} C_VEL
LIN {X 0,Y 159.786,Z 483.64,A -85,B 0,C 180,E1 -24103.387,E2 -24103.387} C_VEL
LIN {X 0,Y 159.26,Z 483.008,A -85,B 0,C 180,E1 -24109.832,E2 -24109.832} C_VEL
LIN {X 0,Y 162.274,Z 484.375,A -85,B 0,C 180,E1 -24120.911,E2 -24120.911} C_VEL
LIN {X 0,Y 163.534,Z 487.504,A -85,B 0,C 180,E1 -24123.715,E2 -24123.715} C_VEL
LIN {X 0,Y 166.234,Z 489.89,A -85,B 0,C 180,E1 -24127.591,E2 -24127.591} C_VEL
LIN {X 0,Y 166.863,Z 490.493,A -85,B 0,C 180,E1 -24128.4,E2 -24128.4} C_VEL
LIN {X 0,Y 168.853,Z 493.861,A -85,B 0,C 180,E1 -24130.912,E2 -24130.912} C_VEL
LIN {X 0,Y 171.05,Z 495.934,A -85,B 0,C 180,E1 -24133.136,E2 -24133.136} C_VEL
LIN {X 0,Y 173.596,Z 499.499,A -85,B 0,C 180,E1 -24135.558,E2 -24135.558} C_VEL
LIN {X 0,Y 174.914,Z 501.049,A -85,B 0,C 180,E1 -24136.68,E2 -24136.68} C_VEL
LIN {X 0,Y 177.738,Z 504.868,A -85,B 0,C 180,E1 -24138.963,E2 -24138.963} C_VEL
LIN {X 0,Y 182.353,Z 511.269,A -85,B 0,C 180,E1 -24142.262,E2 -24142.262} C_VEL
LIN {X 0,Y 187.242,Z 518.28,A -85,B 0,C 180,E1 -24145.338,E2 -24145.338} C_VEL
LIN {X 0,Y 191.219,Z 524.628,A -85,B 0,C 180,E1 -24147.62,E2 -24147.62} C_VEL
LIN {X 0,Y 197.142,Z 536.472,A -85,B 0,C 180,E1 -24150.829,E2 -24150.829} C_VEL
LIN {X 0,Y 202.432,Z 548.069,A -85,B 0,C 180,E1 -24153.438,E2 -24153.438} C_VEL
LIN {X 0,Y 206.851,Z 559.122,A -85,B 0,C 180,E1 -24155.523,E2 -24155.523} C_VEL
LIN {X 0,Y 201.034,Z 631.085,A -85,B 0,C 180,E1 -24157.725,E2 -24157.725} C_VEL
LIN {X 0,Y 198.669,Z 646.756,A -85,B 0,C 180,E1 -24158.493,E2 -24158.493} C_VEL
LIN {X 0,Y 195.409,Z 661.846,A -85,B 0,C 180,E1 -24159.554,E2 -24159.554} C_VEL
LIN {X 0,Y 191.657,Z 675.555,A -85,B 0,C 180,E1 -24160.859,E2 -24160.859} C_VEL
LIN {X 0,Y 188.47,Z 685.349,A -85,B 0,C 180,E1 -24162.046,E2 -24162.046} C_VEL
LIN {X 0,Y 186.237,Z 690.489,A -85,B 0,C 180,E1 -24162.64,E2 -24162.64} C_VEL
LIN {X 0,Y 181.054,Z 698.55,A -85,B 0,C 180,E1 -24163.363,E2 -24163.363} C_VEL
LIN {X 0,Y 175.522,Z 706.349,A -85,B 0,C 180,E1 -24164.215,E2 -24164.215} C_VEL
LIN {X 0,Y 172.77,Z 710.967,A -85,B 0,C 180,E1 -24165.028,E2 -24165.028} C_VEL
LIN {X 0,Y 167.355,Z 722.076,A -85,B 0,C 180,E1 -24167.784,E2 -24167.784} C_VEL
LIN {X 0,Y 161.887,Z 732.32,A -85,B 0,C 180,E1 -24170.987,E2 -24170.987} C_VEL
LIN {X 0,Y 157.121,Z 741.008,A -85,B 0,C 180,E1 -24174.443,E2 -24174.443} C_VEL
LIN {X 0,Y 152.855,Z 748.382,A -85,B 0,C 180,E1 -24178.078,E2 -24178.078} C_VEL
LIN {X 0,Y 148.074,Z 756.56,A -85,B 0,C 180,E1 -24183.197,E2 -24183.197} C_VEL
LIN {X 0,Y 144.502,Z 763.069,A -85,B 0,C 180,E1 -24188.605,E2 -24188.605} C_VEL
LIN {X 0,Y 142.109,Z 768.103,A -85,B 0,C 180,E1 -24194.215,E2 -24194.215} C_VEL
LIN {X 0,Y 141.059,Z 771.018,A -85,B 0,C 180,E1 -24198.503,E2 -24198.503} C_VEL
LIN {X 0,Y 140.518,Z 773.724,A -85,B 0,C 180,E1 -24204.258,E2 -24204.258} C_VEL
LIN {X 0,Y 140.627,Z 775.209,A -85,B 0,C 180,E1 -24209.998,E2 -24209.998} C_VEL
LIN {X 0,Y 140.456,Z 775.503,A -85,B 0,C 180,E1 -24215.742,E2 -24215.742} C_VEL
LIN {X 0,Y 141.067,Z 774.672,A -85,B 0,C 180,E1 -24221.493,E2 -24221.493} C_VEL
LIN {X 0,Y 142.677,Z 772.673,A -85,B 0,C 180,E1 -24227.189,E2 -24227.189} C_VEL
LIN {X 0,Y 145.526,Z 769.517,A -85,B 0,C 180,E1 -24232.726,E2 -24232.726} C_VEL
LIN {X 0,Y 149.607,Z 765.159,A -85,B 0,C 180,E1 -24238.017,E2 -24238.017} C_VEL
LIN {X 0,Y 154.823,Z 759.492,A -85,B 0,C 180,E1 -24243.004,E2 -24243.004} C_VEL
LIN {X 0,Y 161.341,Z 752.377,A -85,B 0,C 180,E1 -24247.575,E2 -24247.575} C_VEL
LIN {X 0,Y 167.472,Z 744.975,A -85,B 0,C 180,E1 -24251.29,E2 -24251.29} C_VEL
LIN {X 0,Y 174.665,Z 735.841,A -85,B 0,C 180,E1 -24254.758,E2 -24254.758} C_VEL
LIN {X 0,Y 182.398,Z 725.019,A -85,B 0,C 180,E1 -24257.876,E2 -24257.876} C_VEL
LIN {X 0,Y 188.167,Z 715.896,A -85,B 0,C 180,E1 -24259.964,E2 -24259.964} C_VEL
LIN {X 0,Y 195.472,Z 703.082,A -85,B 0,C 180,E1 -24262.275,E2 -24262.275} C_VEL
LIN {X 0,Y 201.805,Z 690.181,A -85,B 0,C 180,E1 -24264.064,E2 -24264.064} C_VEL
LIN {X 0,Y 207.03,Z 677.714,A -85,B 0,C 180,E1 -24265.405,E2 -24265.405} C_VEL
LIN {X 0,Y 211.763,Z 664.355,A -85,B 0,C 180,E1 -24266.493,E2 -24266.493} C_VEL
LIN {X 0,Y 215.885,Z 649.7,A -85,B 0,C 180,E1 -24267.385,E2 -24267.385} C_VEL
LIN {X 0,Y 219.038,Z 634.195,A -85,B 0,C 180,E1 -24268.07,E2 -24268.07} C_VEL
LIN {X 0,Y 221.278,Z 616.335,A -85,B 0,C 180,E1 -24268.595,E2 -24268.595} C_VEL
LIN {X 0,Y 225.545,Z 572.954,A -85,B 0,C 180,E1 -24269.725,E2 -24269.725} C_VEL
LIN {X 0,Y 222.941,Z 565.404,A -85,B 0,C 180,E1 -24272.107,E2 -24272.107} C_VEL
LIN {X 0,Y 220.604,Z 559.239,A -85,B 0,C 180,E1 -24274.533,E2 -24274.533} C_VEL
LIN {X 0,Y 218.373,Z 553.828,A -85,B 0,C 180,E1 -24277.282,E2 -24277.282} C_VEL
LIN {X 0,Y 216.386,Z 550.276,A -85,B 0,C 180,E1 -24280.277,E2 -24280.277} C_VEL
LIN {X 0,Y 214.692,Z 546.719,A -85,B 0,C 180,E1 -24284.279,E2 -24284.279} C_VEL
LIN {X 0,Y 214.337,Z 546.262,A -85,B 0,C 180,E1 -24285.472,E2 -24285.472} C_VEL
LIN {X 0,Y 214.058,Z 545.891,A -85,B 0,C 180,E1 -24291.49,E2 -24291.49} C_VEL
LIN {X 0,Y 215.028,Z 546.669,A -85,B 0,C 180,E1 -24294.97,E2 -24294.97} C_VEL
LIN {X 0,Y 216.964,Z 550.718,A -85,B 0,C 180,E1 -24299.044,E2 -24299.044} C_VEL
LIN {X 0,Y 218.928,Z 554.579,A -85,B 0,C 180,E1 -24301.84,E2 -24301.84} C_VEL
LIN {X 0,Y 222.032,Z 560.642,A -85,B 0,C 180,E1 -24305.226,E2 -24305.226} C_VEL
LIN {X 0,Y 225.49,Z 568.22,A -85,B 0,C 180,E1 -24308.293,E2 -24308.293} C_VEL
LIN {X 0,Y 225.806,Z 569.144,A -85,B 0,C 180,E1 -24308.569,E2 -24308.569} C_VEL
LIN {X 0,Y 220.25,Z 624.093,A -85,B 0,C 180,E1 -24310.046,E2 -24310.046} C_VEL
LIN {X 0,Y 217.456,Z 639.784,A -85,B 0,C 180,E1 -24310.681,E2 -24310.681} C_VEL
LIN {X 0,Y 213.94,Z 654.084,A -85,B 0,C 180,E1 -24311.549,E2 -24311.549} C_VEL
LIN {X 0,Y 209.378,Z 668.38,A -85,B 0,C 180,E1 -24312.713,E2 -24312.713} C_VEL
LIN {X 0,Y 203.697,Z 682.733,A -85,B 0,C 180,E1 -24314.253,E2 -24314.253} C_VEL
LIN {X 0,Y 197.469,Z 695.826,A -85,B 0,C 180,E1 -24316.074,E2 -24316.074} C_VEL
LIN {X 0,Y 190.579,Z 708.177,A -85,B 0,C 180,E1 -24318.277,E2 -24318.277} C_VEL
LIN {X 0,Y 184.06,Z 718.6,A -85,B 0,C 180,E1 -24320.698,E2 -24320.698} C_VEL
LIN {X 0,Y 176.596,Z 729.073,A -85,B 0,C 180,E1 -24323.752,E2 -24323.752} C_VEL
LIN {X 0,Y 168.663,Z 739.138,A -85,B 0,C 180,E1 -24327.681,E2 -24327.681} C_VEL
LIN {X 0,Y 162.649,Z 746.056,A -85,B 0,C 180,E1 -24331.233,E2 -24331.233} C_VEL
LIN {X 0,Y 156.148,Z 752.994,A -85,B 0,C 180,E1 -24335.892,E2 -24335.892} C_VEL
LIN {X 0,Y 150.986,Z 758.201,A -85,B 0,C 180,E1 -24340.668,E2 -24340.668} C_VEL
LIN {X 0,Y 146.71,Z 762.314,A -85,B 0,C 180,E1 -24345.937,E2 -24345.937} C_VEL
LIN {X 0,Y 143.505,Z 765.257,A -85,B 0,C 180,E1 -24351.591,E2 -24351.591} C_VEL
LIN {X 0,Y 141.363,Z 767.026,A -85,B 0,C 180,E1 -24357.692,E2 -24357.692} C_VEL
LIN {X 0,Y 140.293,Z 767.525,A -85,B 0,C 180,E1 -24363.203,E2 -24363.203} C_VEL
LIN {X 0,Y 140.066,Z 767.329,A -85,B 0,C 180,E1 -24366.336,E2 -24366.336} C_VEL
LIN {X 0,Y 140.235,Z 765.961,A -85,B 0,C 180,E1 -24372.502,E2 -24372.502} C_VEL
LIN {X 0,Y 141.207,Z 763.323,A -85,B 0,C 180,E1 -24378.518,E2 -24378.518} C_VEL
LIN {X 0,Y 143.122,Z 759.389,A -85,B 0,C 180,E1 -24384.366,E2 -24384.366} C_VEL
LIN {X 0,Y 145.997,Z 754.102,A -85,B 0,C 180,E1 -24390.002,E2 -24390.002} C_VEL
LIN {X 0,Y 149.986,Z 747.32,A -85,B 0,C 180,E1 -24395.379,E2 -24395.379} C_VEL
LIN {X 0,Y 154.318,Z 739.992,A -85,B 0,C 180,E1 -24399.835,E2 -24399.835} C_VEL
LIN {X 0,Y 159.796,Z 730.622,A -85,B 0,C 180,E1 -24404.248,E2 -24404.248} C_VEL
LIN {X 0,Y 165.315,Z 720.52,A -85,B 0,C 180,E1 -24407.953,E2 -24407.953} C_VEL
LIN {X 0,Y 170.873,Z 709.578,A -85,B 0,C 180,E1 -24411.094,E2 -24411.094} C_VEL
LIN {X 0,Y 176.487,Z 697.376,A -85,B 0,C 180,E1 -24413.84,E2 -24413.84} C_VEL
LIN {X 0,Y 181.656,Z 684.538,A -85,B 0,C 180,E1 -24416.11,E2 -24416.11} C_VEL
LIN {X 0,Y 186.521,Z 670.164,A -85,B 0,C 180,E1 -24418.1,E2 -24418.1} C_VEL
LIN {X 0,Y 190.478,Z 656.094,A -85,B 0,C 180,E1 -24419.571,E2 -24419.571} C_VEL
LIN {X 0,Y 193.715,Z 641.196,A -85,B 0,C 180,E1 -24420.753,E2 -24420.753} C_VEL
LIN {X 0,Y 196.252,Z 625.66,A -85,B 0,C 180,E1 -24421.584,E2 -24421.584} C_VEL
LIN {X 0,Y 198.195,Z 605.494,A -85,B 0,C 180,E1 -24422.273,E2 -24422.273} C_VEL
LIN {X 0,Y 202.278,Z 555.458,A -85,B 0,C 180,E1 -24423.774,E2 -24423.774} C_VEL
LIN {X 0,Y 195.211,Z 541.894,A -85,B 0,C 180,E1 -24427.163,E2 -24427.163} C_VEL
LIN {X 0,Y 188.417,Z 530.363,A -85,B 0,C 180,E1 -24430.81,E2 -24430.81} C_VEL
LIN {X 0,Y 182.158,Z 520.657,A -85,B 0,C 180,E1 -24434.655,E2 -24434.655} C_VEL
LIN {X 0,Y 177.99,Z 514.769,A -85,B 0,C 180,E1 -24437.555,E2 -24437.555} C_VEL
LIN {X 0,Y 175.239,Z 510.941,A -85,B 0,C 180,E1 -24439.684,E2 -24439.684} C_VEL
LIN {X 0,Y 172.072,Z 506.598,A -85,B 0,C 180,E1 -24442.407,E2 -24442.407} C_VEL
LIN {X 0,Y 169.237,Z 502.843,A -85,B 0,C 180,E1 -24445.178,E2 -24445.178} C_VEL
LIN {X 0,Y 168.449,Z 501.891,A -85,B 0,C 180,E1 -24446.006,E2 -24446.006} C_VEL
LIN {X 0,Y 166.06,Z 499.165,A -85,B 0,C 180,E1 -24448.758,E2 -24448.758} C_VEL
LIN {X 0,Y 164.968,Z 497.056,A -85,B 0,C 180,E1 -24450.313,E2 -24450.313} C_VEL
LIN {X 0,Y 162.17,Z 494.804,A -85,B 0,C 180,E1 -24454.484,E2 -24454.484} C_VEL
LIN {X 0,Y 160.575,Z 491.509,A -85,B 0,C 180,E1 -24458.159,E2 -24458.159} C_VEL
LIN {X 0,Y 158.337,Z 490.217,A -85,B 0,C 180,E1 -24467.558,E2 -24467.558} C_VEL
LIN {X 0,Y 158.569,Z 490.203,A -85,B 0,C 180,E1 -24472.358,E2 -24472.358} C_VEL
LIN {X 0,Y 161.096,Z 491.405,A -85,B 0,C 180,E1 -24480.434,E2 -24480.434} C_VEL
LIN {X 0,Y 162.329,Z 494.417,A -85,B 0,C 180,E1 -24483.296,E2 -24483.296} C_VEL
LIN {X 0,Y 165.33,Z 497.242,A -85,B 0,C 180,E1 -24487.71,E2 -24487.71} C_VEL
LIN {X 0,Y 167.513,Z 500.795,A -85,B 0,C 180,E1 -24490.546,E2 -24490.546} C_VEL
LIN {X 0,Y 169.367,Z 502.703,A -85,B 0,C 180,E1 -24492.506,E2 -24492.506} C_VEL
LIN {X 0,Y 172.374,Z 506.68,A -85,B 0,C 180,E1 -24495.411,E2 -24495.411} C_VEL
LIN {X 0,Y 175.836,Z 511.436,A -85,B 0,C 180,E1 -24498.343,E2 -24498.343} C_VEL
LIN {X 0,Y 180.097,Z 517.64,A -85,B 0,C 180,E1 -24501.534,E2 -24501.534} C_VEL
LIN {X 0,Y 184.72,Z 524.542,A -85,B 0,C 180,E1 -24504.565,E2 -24504.565} C_VEL
LIN {X 0,Y 187.997,Z 529.888,A -85,B 0,C 180,E1 -24506.547,E2 -24506.547} C_VEL
LIN {X 0,Y 193.524,Z 541.223,A -85,B 0,C 180,E1 -24509.703,E2 -24509.703} C_VEL
LIN {X 0,Y 198.673,Z 552.924,A -85,B 0,C 180,E1 -24512.407,E2 -24512.407} C_VEL
LIN {X 0,Y 202.011,Z 561.528,A -85,B 0,C 180,E1 -24514.073,E2 -24514.073} C_VEL
LIN {X 0,Y 196.247,Z 630.709,A -85,B 0,C 180,E1 -24516.206,E2 -24516.206} C_VEL
LIN {X 0,Y 193.833,Z 646.446,A -85,B 0,C 180,E1 -24516.983,E2 -24516.983} C_VEL
LIN {X 0,Y 190.624,Z 660.992,A -85,B 0,C 180,E1 -24517.994,E2 -24517.994} C_VEL
LIN {X 0,Y 186.457,Z 675.739,A -85,B 0,C 180,E1 -24519.403,E2 -24519.403} C_VEL
LIN {X 0,Y 182.059,Z 688.757,A -85,B 0,C 180,E1 -24521.055,E2 -24521.055} C_VEL
LIN {X 0,Y 176.894,Z 701.56,A -85,B 0,C 180,E1 -24523.109,E2 -24523.109} C_VEL
LIN {X 0,Y 172.77,Z 710.967,A -85,B 0,C 180,E1 -24525.028,E2 -24525.028} C_VEL
LIN {X 0,Y 169.971,Z 715.514,A -85,B 0,C 180,E1 -24525.904,E2 -24525.904} C_VEL
LIN {X 0,Y 164.03,Z 722.56,A -85,B 0,C 180,E1 -24527.168,E2 -24527.168} C_VEL
LIN {X 0,Y 158.12,Z 729.26,A -85,B 0,C 180,E1 -24528.676,E2 -24528.676} C_VEL
LIN {X 0,Y 155.396,Z 733.155,A -85,B 0,C 180,E1 -24529.948,E2 -24529.948} C_VEL
LIN {X 0,Y 150.519,Z 741.615,A -85,B 0,C 180,E1 -24533.463,E2 -24533.463} C_VEL
LIN {X 0,Y 145.369,Z 749.998,A -85,B 0,C 180,E1 -24537.871,E2 -24537.871} C_VEL
LIN {X 0,Y 140.608,Z 757.831,A -85,B 0,C 180,E1 -24543.265,E2 -24543.265} C_VEL
LIN {X 0,Y 137.051,Z 764.027,A -85,B 0,C 180,E1 -24548.962,E2 -24548.962} C_VEL
LIN {X 0,Y 134.728,Z 768.768,A -85,B 0,C 180,E1 -24554.88,E2 -24554.88} C_VEL
LIN {X 0,Y 133.601,Z 772.176,A -85,B 0,C 180,E1 -24560.918,E2 -24560.918} C_VEL
LIN {X 0,Y 133.394,Z 774.329,A -85,B 0,C 180,E1 -24566.978,E2 -24566.978} C_VEL
LIN {X 0,Y 133.53,Z 774.954,A -85,B 0,C 180,E1 -24569.998,E2 -24569.998} C_VEL
LIN {X 0,Y 133.386,Z 775.31,A -85,B 0,C 180,E1 -24576.047,E2 -24576.047} C_VEL
LIN {X 0,Y 134.065,Z 774.535,A -85,B 0,C 180,E1 -24582.102,E2 -24582.102} C_VEL
LIN {X 0,Y 135.841,Z 772.582,A -85,B 0,C 180,E1 -24588.083,E2 -24588.083} C_VEL
LIN {X 0,Y 139.766,Z 768.662,A -85,B 0,C 180,E1 -24595.163,E2 -24595.163} C_VEL
LIN {X 0,Y 144.614,Z 763.963,A -85,B 0,C 180,E1 -24600.68,E2 -24600.68} C_VEL
LIN {X 0,Y 150.524,Z 758.029,A -85,B 0,C 180,E1 -24605.704,E2 -24605.704} C_VEL
LIN {X 0,Y 156.989,Z 751.183,A -85,B 0,C 180,E1 -24610.008,E2 -24610.008} C_VEL
LIN {X 0,Y 163.29,Z 743.987,A -85,B 0,C 180,E1 -24613.52,E2 -24613.52} C_VEL
LIN {X 0,Y 170.816,Z 734.85,A -85,B 0,C 180,E1 -24616.909,E2 -24616.909} C_VEL
LIN {X 0,Y 177.739,Z 725.614,A -85,B 0,C 180,E1 -24619.564,E2 -24619.564} C_VEL
LIN {X 0,Y 183.712,Z 716.648,A -85,B 0,C 180,E1 -24621.647,E2 -24621.647} C_VEL
LIN {X 0,Y 191.252,Z 704.037,A -85,B 0,C 180,E1 -24623.941,E2 -24623.941} C_VEL
LIN {X 0,Y 197.769,Z 691.383,A -85,B 0,C 180,E1 -24625.71,E2 -24625.71} C_VEL
LIN {X 0,Y 203.832,Z 677.514,A -85,B 0,C 180,E1 -24627.183,E2 -24627.183} C_VEL
LIN {X 0,Y 208.695,Z 664.156,A -85,B 0,C 180,E1 -24628.243,E2 -24628.243} C_VEL
LIN {X 0,Y 212.92,Z 649.565,A -85,B 0,C 180,E1 -24629.112,E2 -24629.112} C_VEL
LIN {X 0,Y 216.097,Z 634.534,A -85,B 0,C 180,E1 -24629.765,E2 -24629.765} C_VEL
LIN {X 0,Y 218.372,Z 617.352,A -85,B 0,C 180,E1 -24630.269,E2 -24630.269} C_VEL
LIN {X 0,Y 222.541,Z 576.382,A -85,B 0,C 180,E1 -24631.327,E2 -24631.327} C_VEL
LIN {X 0,Y 220.183,Z 569.134,A -85,B 0,C 180,E1 -24633.757,E2 -24633.757} C_VEL
LIN {X 0,Y 218.137,Z 563.495,A -85,B 0,C 180,E1 -24636.217,E2 -24636.217} C_VEL
LIN {X 0,Y 216.763,Z 560.179,A -85,B 0,C 180,E1 -24638.108,E2 -24638.108} C_VEL
LIN {X 0,Y 215.243,Z 557.185,A -85,B 0,C 180,E1 -24640.587,E2 -24640.587} C_VEL
LIN {X 0,Y 213.524,Z 553.344,A -85,B 0,C 180,E1 -24645.075,E2 -24645.075} C_VEL
LIN {X 0,Y 213.141,Z 552.942,A -85,B 0,C 180,E1 -24651.562,E2 -24651.562} C_VEL
LIN {X 0,Y 213.988,Z 553.713,A -85,B 0,C 180,E1 -24654.728,E2 -24654.728} C_VEL
LIN {X 0,Y 215.791,Z 557.732,A -85,B 0,C 180,E1 -24658.741,E2 -24658.741} C_VEL
LIN {X 0,Y 217.503,Z 561.292,A -85,B 0,C 180,E1 -24661.333,E2 -24661.333} C_VEL
LIN {X 0,Y 220.244,Z 566.927,A -85,B 0,C 180,E1 -24664.506,E2 -24664.506} C_VEL
LIN {X 0,Y 222.818,Z 572.909,A -85,B 0,C 180,E1 -24666.991,E2 -24666.991} C_VEL
LIN {X 0,Y 217.442,Z 624.093,A -85,B 0,C 180,E1 -24668.339,E2 -24668.339} C_VEL
LIN {X 0,Y 214.468,Z 640.281,A -85,B 0,C 180,E1 -24668.984,E2 -24668.984} C_VEL
LIN {X 0,Y 211.096,Z 653.552,A -85,B 0,C 180,E1 -24669.762,E2 -24669.762} C_VEL
LIN {X 0,Y 206.623,Z 667.349,A -85,B 0,C 180,E1 -24670.854,E2 -24670.854} C_VEL
LIN {X 0,Y 201.328,Z 680.634,A -85,B 0,C 180,E1 -24672.205,E2 -24672.205} C_VEL
LIN {X 0,Y 195.404,Z 693.078,A -85,B 0,C 180,E1 -24673.816,E2 -24673.816} C_VEL
LIN {X 0,Y 188.231,Z 705.955,A -85,B 0,C 180,E1 -24675.972,E2 -24675.972} C_VEL
LIN {X 0,Y 180.865,Z 717.452,A -85,B 0,C 180,E1 -24678.495,E2 -24678.495} C_VEL
LIN {X 0,Y 173.283,Z 727.802,A -85,B 0,C 180,E1 -24681.41,E2 -24681.41} C_VEL
LIN {X 0,Y 166.581,Z 736.111,A -85,B 0,C 180,E1 -24684.447,E2 -24684.447} C_VEL
LIN {X 0,Y 159.505,Z 744.115,A -85,B 0,C 180,E1 -24688.213,E2 -24688.213} C_VEL
LIN {X 0,Y 153.397,Z 750.42,A -85,B 0,C 180,E1 -24692.053,E2 -24692.053} C_VEL
LIN {X 0,Y 148.07,Z 755.57,A -85,B 0,C 180,E1 -24696.21,E2 -24696.21} C_VEL
LIN {X 0,Y 143.535,Z 759.763,A -85,B 0,C 180,E1 -24700.632,E2 -24700.632} C_VEL
LIN {X 0,Y 139.846,Z 762.986,A -85,B 0,C 180,E1 -24705.288,E2 -24705.288} C_VEL
LIN {X 0,Y 136.234,Z 765.956,A -85,B 0,C 180,E1 -24711.756,E2 -24711.756} C_VEL
LIN {X 0,Y 134.05,Z 767.467,A -85,B 0,C 180,E1 -24718.382,E2 -24718.382} C_VEL
LIN {X 0,Y 133.029,Z 767.6,A -85,B 0,C 180,E1 -24725.001,E2 -24725.001} C_VEL
LIN {X 0,Y 133.042,Z 766.419,A -85,B 0,C 180,E1 -24731.523,E2 -24731.523} C_VEL
LIN {X 0,Y 133.933,Z 763.969,A -85,B 0,C 180,E1 -24737.886,E2 -24737.886} C_VEL
LIN {X 0,Y 135.812,Z 760.228,A -85,B 0,C 180,E1 -24744.061,E2 -24744.061} C_VEL
LIN {X 0,Y 138.717,Z 755.141,A -85,B 0,C 180,E1 -24750.002,E2 -24750.002} C_VEL
LIN {X 0,Y 142.745,Z 748.579,A -85,B 0,C 180,E1 -24755.653,E2 -24755.653} C_VEL
LIN {X 0,Y 147.176,Z 741.49,A -85,B 0,C 180,E1 -24760.317,E2 -24760.317} C_VEL
LIN {X 0,Y 152.682,Z 732.563,A -85,B 0,C 180,E1 -24764.839,E2 -24764.839} C_VEL
LIN {X 0,Y 158.445,Z 722.588,A -85,B 0,C 180,E1 -24768.76,E2 -24768.76} C_VEL
LIN {X 0,Y 164.136,Z 712.011,A -85,B 0,C 180,E1 -24772.004,E2 -24772.004} C_VEL
LIN {X 0,Y 169.923,Z 700.214,A -85,B 0,C 180,E1 -24774.828,E2 -24774.828} C_VEL
LIN {X 0,Y 175.2,Z 687.952,A -85,B 0,C 180,E1 -24777.15,E2 -24777.15} C_VEL
LIN {X 0,Y 180.247,Z 674.284,A -85,B 0,C 180,E1 -24779.17,E2 -24779.17} C_VEL
LIN {X 0,Y 184.568,Z 660.16,A -85,B 0,C 180,E1 -24780.776,E2 -24780.776} C_VEL
LIN {X 0,Y 188.136,Z 645.667,A -85,B 0,C 180,E1 -24782.006,E2 -24782.006} C_VEL
LIN {X 0,Y 190.984,Z 630.067,A -85,B 0,C 180,E1 -24782.953,E2 -24782.953} C_VEL
LIN {X 0,Y 192.853,Z 614.073,A -85,B 0,C 180,E1 -24783.577,E2 -24783.577} C_VEL
LIN {X 0,Y 197.536,Z 558.887,A -85,B 0,C 180,E1 -24785.226,E2 -24785.226} C_VEL
LIN {X 0,Y 197.227,Z 557.691,A -85,B 0,C 180,E1 -24785.411,E2 -24785.411} C_VEL
LIN {X 0,Y 190.576,Z 544.828,A -85,B 0,C 180,E1 -24788.859,E2 -24788.859} C_VEL
LIN {X 0,Y 184.187,Z 533.9,A -85,B 0,C 180,E1 -24792.568,E2 -24792.568} C_VEL
LIN {X 0,Y 178.858,Z 525.505,A -85,B 0,C 180,E1 -24796.085,E2 -24796.085} C_VEL
LIN {X 0,Y 175.004,Z 519.974,A -85,B 0,C 180,E1 -24798.968,E2 -24798.968} C_VEL
LIN {X 0,Y 172.802,Z 516.876,A -85,B 0,C 180,E1 -24800.772,E2 -24800.772} C_VEL
LIN {X 0,Y 170.114,Z 513.006,A -85,B 0,C 180,E1 -24803.237,E2 -24803.237} C_VEL
LIN {X 0,Y 167.261,Z 508.984,A -85,B 0,C 180,E1 -24806.187,E2 -24806.187} C_VEL
LIN {X 0,Y 164.498,Z 505.761,A -85,B 0,C 180,E1 -24809.49,E2 -24809.49} C_VEL
LIN {X 0,Y 163.419,Z 503.812,A -85,B 0,C 180,E1 -24811.064,E2 -24811.064} C_VEL
LIN {X 0,Y 160.843,Z 501.52,A -85,B 0,C 180,E1 -24815.179,E2 -24815.179} C_VEL
LIN {X 0,Y 159.417,Z 498.464,A -85,B 0,C 180,E1 -24818.671,E2 -24818.671} C_VEL
LIN {X 0,Y 157.41,Z 497.089,A -85,B 0,C 180,E1 -24829.712,E2 -24829.712} C_VEL
LIN {X 0,Y 159.868,Z 498.277,A -85,B 0,C 180,E1 -24839.81,E2 -24839.81} C_VEL
LIN {X 0,Y 161.117,Z 501.295,A -85,B 0,C 180,E1 -24842.837,E2 -24842.837} C_VEL
LIN {X 0,Y 163.855,Z 504.071,A -85,B 0,C 180,E1 -24847.083,E2 -24847.083} C_VEL
LIN {X 0,Y 166.184,Z 507.723,A -85,B 0,C 180,E1 -24850.185,E2 -24850.185} C_VEL
LIN {X 0,Y 167.639,Z 509.304,A -85,B 0,C 180,E1 -24851.782,E2 -24851.782} C_VEL
LIN {X 0,Y 171.055,Z 514.132,A -85,B 0,C 180,E1 -24855.217,E2 -24855.217} C_VEL
LIN {X 0,Y 174.647,Z 519.289,A -85,B 0,C 180,E1 -24858.309,E2 -24858.309} C_VEL
LIN {X 0,Y 177.843,Z 523.97,A -85,B 0,C 180,E1 -24860.767,E2 -24860.767} C_VEL
LIN {X 0,Y 182.685,Z 531.453,A -85,B 0,C 180,E1 -24864.06,E2 -24864.06} C_VEL
LIN {X 0,Y 185.182,Z 535.791,A -85,B 0,C 180,E1 -24865.65,E2 -24865.65} C_VEL
LIN {X 0,Y 190.341,Z 546.867,A -85,B 0,C 180,E1 -24868.76,E2 -24868.76} C_VEL
LIN {X 0,Y 195.008,Z 557.843,A -85,B 0,C 180,E1 -24871.353,E2 -24871.353} C_VEL
LIN {X 0,Y 197.331,Z 564.035,A -85,B 0,C 180,E1 -24872.593,E2 -24872.593} C_VEL
LIN {X 0,Y 191.567,Z 630.345,A -85,B 0,C 180,E1 -24874.622,E2 -24874.622} C_VEL
LIN {X 0,Y 189.115,Z 645.972,A -85,B 0,C 180,E1 -24875.387,E2 -24875.387} C_VEL
LIN {X 0,Y 185.674,Z 661.165,A -85,B 0,C 180,E1 -24876.453,E2 -24876.453} C_VEL
LIN {X 0,Y 181.986,Z 673.93,A -85,B 0,C 180,E1 -24877.656,E2 -24877.656} C_VEL
LIN {X 0,Y 177.152,Z 687.949,A -85,B 0,C 180,E1 -24879.401,E2 -24879.401} C_VEL
LIN {X 0,Y 172.109,Z 700.289,A -85,B 0,C 180,E1 -24881.38,E2 -24881.38} C_VEL
LIN {X 0,Y 166.671,Z 712.027,A -85,B 0,C 180,E1 -24883.77,E2 -24883.77} C_VEL
LIN {X 0,Y 161.105,Z 722.945,A -85,B 0,C 180,E1 -24886.6,E2 -24886.6} C_VEL
LIN {X 0,Y 155.396,Z 733.155,A -85,B 0,C 180,E1 -24889.948,E2 -24889.948} C_VEL
LIN {X 0,Y 152.657,Z 736.98,A -85,B 0,C 180,E1 -24891.31,E2 -24891.31} C_VEL
LIN {X 0,Y 146.647,Z 742.751,A -85,B 0,C 180,E1 -24893.362,E2 -24893.362} C_VEL
LIN {X 0,Y 140.686,Z 748.135,A -85,B 0,C 180,E1 -24895.7,E2 -24895.7} C_VEL
LIN {X 0,Y 138.107,Z 751.19,A -85,B 0,C 180,E1 -24897.495,E2 -24897.495} C_VEL
LIN {X 0,Y 133.118,Z 758.923,A -85,B 0,C 180,E1 -24903.336,E2 -24903.336} C_VEL
LIN {X 0,Y 129.64,Z 764.833,A -85,B 0,C 180,E1 -24909.366,E2 -24909.366} C_VEL
LIN {X 0,Y 127.824,Z 768.331,A -85,B 0,C 180,E1 -24914.042,E2 -24914.042} C_VEL
LIN {X 0,Y 126.56,Z 771.813,A -85,B 0,C 180,E1 -24920.409,E2 -24920.409} C_VEL
LIN {X 0,Y 126.298,Z 774.036,A -85,B 0,C 180,E1 -24926.808,E2 -24926.808} C_VEL
LIN {X 0,Y 126.443,Z 774.696,A -85,B 0,C 180,E1 -24929.998,E2 -24929.998} C_VEL
LIN {X 0,Y 126.293,Z 775.117,A -85,B 0,C 180,E1 -24936.388,E2 -24936.388} C_VEL
LIN {X 0,Y 127.065,Z 774.378,A -85,B 0,C 180,E1 -24942.78,E2 -24942.78} C_VEL
LIN {X 0,Y 129.048,Z 772.49,A -85,B 0,C 180,E1 -24949.07,E2 -24949.07} C_VEL
LIN {X 0,Y 133.01,Z 768.905,A -85,B 0,C 180,E1 -24956.073,E2 -24956.073} C_VEL
LIN {X 0,Y 138.509,Z 764.041,A -85,B 0,C 180,E1 -24962.191,E2 -24962.191} C_VEL
LIN {X 0,Y 144.793,Z 758.191,A -85,B 0,C 180,E1 -24967.351,E2 -24967.351} C_VEL
LIN {X 0,Y 151.397,Z 751.636,A -85,B 0,C 180,E1 -24971.636,E2 -24971.636} C_VEL
LIN {X 0,Y 158.21,Z 744.375,A -85,B 0,C 180,E1 -24975.293,E2 -24975.293} C_VEL
LIN {X 0,Y 166.064,Z 735.38,A -85,B 0,C 180,E1 -24978.691,E2 -24978.691} C_VEL
LIN {X 0,Y 174.458,Z 724.587,A -85,B 0,C 180,E1 -24981.769,E2 -24981.769} C_VEL
LIN {X 0,Y 182.006,Z 713.562,A -85,B 0,C 180,E1 -24984.18,E2 -24984.18} C_VEL
LIN {X 0,Y 189.623,Z 700.848,A -85,B 0,C 180,E1 -24986.308,E2 -24986.308} C_VEL
LIN {X 0,Y 195.995,Z 688.448,A -85,B 0,C 180,E1 -24987.899,E2 -24987.899} C_VEL
LIN {X 0,Y 201.519,Z 675.733,A -85,B 0,C 180,E1 -24989.179,E2 -24989.179} C_VEL
LIN {X 0,Y 206.544,Z 661.984,A -85,B 0,C 180,E1 -24990.187,E2 -24990.187} C_VEL
LIN {X 0,Y 210.801,Z 647.119,A -85,B 0,C 180,E1 -24990.992,E2 -24990.992} C_VEL
LIN {X 0,Y 213.804,Z 632.523,A -85,B 0,C 180,E1 -24991.578,E2 -24991.578} C_VEL
LIN {X 0,Y 216.291,Z 612.674,A -85,B 0,C 180,E1 -24992.134,E2 -24992.134} C_VEL
LIN {X 0,Y 219.747,Z 579.868,A -85,B 0,C 180,E1 -24992.952,E2 -24992.952} C_VEL
LIN {X 0,Y 217.476,Z 572.514,A -85,B 0,C 180,E1 -24995.683,E2 -24995.683} C_VEL
LIN {X 0,Y 215.522,Z 567.05,A -85,B 0,C 180,E1 -24998.479,E2 -24998.479} C_VEL
LIN {X 0,Y 213.943,Z 563.864,A -85,B 0,C 180,E1 -25001.198,E2 -25001.198} C_VEL
LIN {X 0,Y 212.512,Z 560.337,A -85,B 0,C 180,E1 -25005.344,E2 -25005.344} C_VEL
LIN {X 0,Y 212.197,Z 559.973,A -85,B 0,C 180,E1 -25011.472,E2 -25011.472} C_VEL
LIN {X 0,Y 212.944,Z 560.689,A -85,B 0,C 180,E1 -25014.446,E2 -25014.446} C_VEL
LIN {X 0,Y 214.586,Z 564.578,A -85,B 0,C 180,E1 -25018.352,E2 -25018.352} C_VEL
LIN {X 0,Y 216.123,Z 568.032,A -85,B 0,C 180,E1 -25020.83,E2 -25020.83} C_VEL
LIN {X 0,Y 218.763,Z 573.864,A -85,B 0,C 180,E1 -25024.071,E2 -25024.071} C_VEL
LIN {X 0,Y 219.945,Z 576.855,A -85,B 0,C 180,E1 -25025.351,E2 -25025.351} C_VEL
LIN {X 0,Y 214.859,Z 624.09,A -85,B 0,C 180,E1 -25026.585,E2 -25026.585} C_VEL
LIN {X 0,Y 211.952,Z 639.777,A -85,B 0,C 180,E1 -25027.184,E2 -25027.184} C_VEL
LIN {X 0,Y 207.972,Z 654.928,A -85,B 0,C 180,E1 -25028.05,E2 -25028.05} C_VEL
LIN {X 0,Y 203.306,Z 668.68,A -85,B 0,C 180,E1 -25029.13,E2 -25029.13} C_VEL
LIN {X 0,Y 197.325,Z 682.919,A -85,B 0,C 180,E1 -25030.593,E2 -25030.593} C_VEL
LIN {X 0,Y 190.752,Z 695.897,A -85,B 0,C 180,E1 -25032.327,E2 -25032.327} C_VEL
LIN {X 0,Y 183.277,Z 708.425,A -85,B 0,C 180,E1 -25034.486,E2 -25034.486} C_VEL
LIN {X 0,Y 176.211,Z 718.815,A -85,B 0,C 180,E1 -25036.828,E2 -25036.828} C_VEL
LIN {X 0,Y 167.73,Z 729.772,A -85,B 0,C 180,E1 -25040.002,E2 -25040.002} C_VEL
LIN {X 0,Y 159.356,Z 739.388,A -85,B 0,C 180,E1 -25043.781,E2 -25043.781} C_VEL
LIN {X 0,Y 151.394,Z 747.553,A -85,B 0,C 180,E1 -25048.118,E2 -25048.118} C_VEL
LIN {X 0,Y 145.293,Z 753.235,A -85,B 0,C 180,E1 -25052.147,E2 -25052.147} C_VEL
LIN {X 0,Y 139.204,Z 758.588,A -85,B 0,C 180,E1 -25057.291,E2 -25057.291} C_VEL
LIN {X 0,Y 134.15,Z 762.712,A -85,B 0,C 180,E1 -25062.928,E2 -25062.928} C_VEL
LIN {X 0,Y 130.012,Z 765.836,A -85,B 0,C 180,E1 -25069.561,E2 -25069.561} C_VEL
LIN {X 0,Y 127.392,Z 767.545,A -85,B 0,C 180,E1 -25076.52,E2 -25076.52} C_VEL
LIN {X 0,Y 126.075,Z 767.87,A -85,B 0,C 180,E1 -25083.518,E2 -25083.518} C_VEL
LIN {X 0,Y 125.859,Z 766.876,A -85,B 0,C 180,E1 -25090.427,E2 -25090.427} C_VEL
LIN {X 0,Y 126.669,Z 764.606,A -85,B 0,C 180,E1 -25097.179,E2 -25097.179} C_VEL
LIN {X 0,Y 128.489,Z 761.054,A -85,B 0,C 180,E1 -25103.721,E2 -25103.721} C_VEL
LIN {X 0,Y 131.42,Z 756.161,A -85,B 0,C 180,E1 -25110.002,E2 -25110.002} C_VEL
LIN {X 0,Y 135.523,Z 749.811,A -85,B 0,C 180,E1 -25115.955,E2 -25115.955} C_VEL
LIN {X 0,Y 140.761,Z 741.815,A -85,B 0,C 180,E1 -25121.522,E2 -25121.522} C_VEL
LIN {X 0,Y 146.151,Z 733.561,A -85,B 0,C 180,E1 -25125.896,E2 -25125.896} C_VEL
LIN {X 0,Y 151.649,Z 724.563,A -85,B 0,C 180,E1 -25129.634,E2 -25129.634} C_VEL
LIN {X 0,Y 157.486,Z 714.281,A -85,B 0,C 180,E1 -25132.986,E2 -25132.986} C_VEL
LIN {X 0,Y 163.533,Z 702.596,A -85,B 0,C 180,E1 -25135.957,E2 -25135.957} C_VEL
LIN {X 0,Y 168.833,Z 691.049,A -85,B 0,C 180,E1 -25138.263,E2 -25138.263} C_VEL
LIN {X 0,Y 174.034,Z 678.01,A -85,B 0,C 180,E1 -25140.318,E2 -25140.318} C_VEL
LIN {X 0,Y 178.757,Z 663.767,A -85,B 0,C 180,E1 -25142.058,E2 -25142.058} C_VEL
LIN {X 0,Y 182.72,Z 648.984,A -85,B 0,C 180,E1 -25143.403,E2 -25143.403} C_VEL
LIN {X 0,Y 185.605,Z 634.699,A -85,B 0,C 180,E1 -25144.364,E2 -25144.364} C_VEL
LIN {X 0,Y 187.849,Z 618.973,A -85,B 0,C 180,E1 -25145.054,E2 -25145.054} C_VEL
LIN {X 0,Y 192.943,Z 561.962,A -85,B 0,C 180,E1 -25146.768,E2 -25146.768} C_VEL
LIN {X 0,Y 192.686,Z 560.683,A -85,B 0,C 180,E1 -25146.951,E2 -25146.951} C_VEL
LIN {X 0,Y 186.85,Z 549.304,A -85,B 0,C 180,E1 -25150.167,E2 -25150.167} C_VEL
LIN {X 0,Y 181.212,Z 539.358,A -85,B 0,C 180,E1 -25153.652,E2 -25153.652} C_VEL
LIN {X 0,Y 176.164,Z 531.164,A -85,B 0,C 180,E1 -25157.188,E2 -25157.188} C_VEL
LIN {X 0,Y 171.343,Z 523.903,A -85,B 0,C 180,E1 -25161.093,E2 -25161.093} C_VEL
LIN {X 0,Y 167.996,Z 519.17,A -85,B 0,C 180,E1 -25164.271,E2 -25164.271} C_VEL
LIN {X 0,Y 165.315,Z 515.296,A -85,B 0,C 180,E1 -25167.214,E2 -25167.214} C_VEL
LIN {X 0,Y 162.808,Z 512.107,A -85,B 0,C 180,E1 -25170.436,E2 -25170.436} C_VEL
LIN {X 0,Y 161.829,Z 510.511,A -85,B 0,C 180,E1 -25171.925,E2 -25171.925} C_VEL
LIN {X 0,Y 159.437,Z 508.051,A -85,B 0,C 180,E1 -25176.092,E2 -25176.092} C_VEL
LIN {X 0,Y 158.266,Z 505.44,A -85,B 0,C 180,E1 -25179.191,E2 -25179.191} C_VEL
LIN {X 0,Y 156.486,Z 504.12,A -85,B 0,C 180,E1 -25189.65,E2 -25189.65} C_VEL
LIN {X 0,Y 158.701,Z 505.313,A -85,B 0,C 180,E1 -25199.333,E2 -25199.333} C_VEL
LIN {X 0,Y 160.072,Z 508.411,A -85,B 0,C 180,E1 -25202.685,E2 -25202.685} C_VEL
LIN {X 0,Y 162.395,Z 510.819,A -85,B 0,C 180,E1 -25206.434,E2 -25206.434} C_VEL
LIN {X 0,Y 164.738,Z 514.516,A -85,B 0,C 180,E1 -25209.67,E2 -25209.67} C_VEL
LIN {X 0,Y 166.043,Z 516.08,A -85,B 0,C 180,E1 -25211.179,E2 -25211.179} C_VEL
LIN {X 0,Y 169.15,Z 520.584,A -85,B 0,C 180,E1 -25214.435,E2 -25214.435} C_VEL
LIN {X 0,Y 172.802,Z 526.033,A -85,B 0,C 180,E1 -25217.731,E2 -25217.731} C_VEL
LIN {X 0,Y 176.765,Z 531.971,A -85,B 0,C 180,E1 -25220.833,E2 -25220.833} C_VEL
LIN {X 0,Y 181.783,Z 540.358,A -85,B 0,C 180,E1 -25224.298,E2 -25224.298} C_VEL
LIN {X 0,Y 186.858,Z 551.675,A -85,B 0,C 180,E1 -25227.586,E2 -25227.586} C_VEL
LIN {X 0,Y 191.312,Z 562.538,A -85,B 0,C 180,E1 -25230.205,E2 -25230.205} C_VEL
LIN {X 0,Y 192.71,Z 566.334,A -85,B 0,C 180,E1 -25231.005,E2 -25231.005} C_VEL
LIN {X 0,Y 186.948,Z 630.552,A -85,B 0,C 180,E1 -25232.992,E2 -25232.992} C_VEL
LIN {X 0,Y 184.404,Z 646.173,A -85,B 0,C 180,E1 -25233.765,E2 -25233.765} C_VEL
LIN {X 0,Y 180.858,Z 661.259,A -85,B 0,C 180,E1 -25234.824,E2 -25234.824} C_VEL
LIN {X 0,Y 177.07,Z 673.993,A -85,B 0,C 180,E1 -25236.03,E2 -25236.03} C_VEL
LIN {X 0,Y 171.999,Z 688.143,A -85,B 0,C 180,E1 -25237.8,E2 -25237.8} C_VEL
LIN {X 0,Y 166.867,Z 700.259,A -85,B 0,C 180,E1 -25239.766,E2 -25239.766} C_VEL
LIN {X 0,Y 161.239,Z 711.97,A -85,B 0,C 180,E1 -25242.183,E2 -25242.183} C_VEL
LIN {X 0,Y 155.973,Z 721.959,A -85,B 0,C 180,E1 -25244.79,E2 -25244.79} C_VEL
LIN {X 0,Y 150.031,Z 732.159,A -85,B 0,C 180,E1 -25248.123,E2 -25248.123} C_VEL
LIN {X 0,Y 144.798,Z 740.83,A -85,B 0,C 180,E1 -25251.767,E2 -25251.767} C_VEL
LIN {X 0,Y 140.11,Z 748.169,A -85,B 0,C 180,E1 -25255.644,E2 -25255.644} C_VEL
LIN {X 0,Y 138.107,Z 751.19,A -85,B 0,C 180,E1 -25257.495,E2 -25257.495} C_VEL
LIN {X 0,Y 135.627,Z 754.13,A -85,B 0,C 180,E1 -25259.39,E2 -25259.39} C_VEL
LIN {X 0,Y 130.103,Z 758.418,A -85,B 0,C 180,E1 -25262.412,E2 -25262.412} C_VEL
LIN {X 0,Y 124.868,Z 762.265,A -85,B 0,C 180,E1 -25265.789,E2 -25265.789} C_VEL
LIN {X 0,Y 122.93,Z 764.355,A -85,B 0,C 180,E1 -25268.186,E2 -25268.186} C_VEL
LIN {X 0,Y 120.95,Z 767.891,A -85,B 0,C 180,E1 -25273.108,E2 -25273.108} C_VEL
LIN {X 0,Y 119.54,Z 771.449,A -85,B 0,C 180,E1 -25279.839,E2 -25279.839} C_VEL
LIN {X 0,Y 119.212,Z 773.743,A -85,B 0,C 180,E1 -25286.618,E2 -25286.618} C_VEL
LIN {X 0,Y 119.358,Z 774.437,A -85,B 0,C 180,E1 -25289.998,E2 -25289.998} C_VEL
LIN {X 0,Y 119.216,Z 774.922,A -85,B 0,C 180,E1 -25296.769,E2 -25296.769} C_VEL
LIN {X 0,Y 120.096,Z 774.221,A -85,B 0,C 180,E1 -25303.535,E2 -25303.535} C_VEL
LIN {X 0,Y 122.304,Z 772.411,A -85,B 0,C 180,E1 -25310.166,E2 -25310.166} C_VEL
LIN {X 0,Y 126.35,Z 769.119,A -85,B 0,C 180,E1 -25317.132,E2 -25317.132} C_VEL
LIN {X 0,Y 131.039,Z 765.37,A -85,B 0,C 180,E1 -25322.432,E2 -25322.432} C_VEL
LIN {X 0,Y 137.355,Z 759.982,A -85,B 0,C 180,E1 -25327.877,E2 -25327.877} C_VEL
LIN {X 0,Y 144.942,Z 753.166,A -85,B 0,C 180,E1 -25332.75,E2 -25332.75} C_VEL
LIN {X 0,Y 151.115,Z 746.991,A -85,B 0,C 180,E1 -25336.124,E2 -25336.124} C_VEL
LIN {X 0,Y 159.079,Z 738.542,A -85,B 0,C 180,E1 -25339.646,E2 -25339.646} C_VEL
LIN {X 0,Y 167.657,Z 728.445,A -85,B 0,C 180,E1 -25342.79,E2 -25342.79} C_VEL
LIN {X 0,Y 175.329,Z 718.228,A -85,B 0,C 180,E1 -25345.256,E2 -25345.256} C_VEL
LIN {X 0,Y 183.335,Z 706.062,A -85,B 0,C 180,E1 -25347.492,E2 -25347.492} C_VEL
LIN {X 0,Y 190.238,Z 693.957,A -85,B 0,C 180,E1 -25349.193,E2 -25349.193} C_VEL
LIN {X 0,Y 196.616,Z 680.794,A -85,B 0,C 180,E1 -25350.604,E2 -25350.604} C_VEL
LIN {X 0,Y 202.434,Z 666.325,A -85,B 0,C 180,E1 -25351.754,E2 -25351.754} C_VEL
LIN {X 0,Y 207.227,Z 651.204,A -85,B 0,C 180,E1 -25352.633,E2 -25352.633} C_VEL
LIN {X 0,Y 210.903,Z 635.308,A -85,B 0,C 180,E1 -25353.297,E2 -25353.297} C_VEL
LIN {X 0,Y 213.265,Z 619.295,A -85,B 0,C 180,E1 -25353.749,E2 -25353.749} C_VEL
LIN {X 0,Y 217.143,Z 583.522,A -85,B 0,C 180,E1 -25354.637,E2 -25354.637} C_VEL
LIN {X 0,Y 215.447,Z 577.714,A -85,B 0,C 180,E1 -25356.956,E2 -25356.956} C_VEL
LIN {X 0,Y 213.963,Z 573.305,A -85,B 0,C 180,E1 -25359.374,E2 -25359.374} C_VEL
LIN {X 0,Y 212.834,Z 570.78,A -85,B 0,C 180,E1 -25361.509,E2 -25361.509} C_VEL
LIN {X 0,Y 211.519,Z 567.348,A -85,B 0,C 180,E1 -25365.594,E2 -25365.594} C_VEL
LIN {X 0,Y 211.262,Z 567.01,A -85,B 0,C 180,E1 -25371.434,E2 -25371.434} C_VEL
LIN {X 0,Y 211.916,Z 567.726,A -85,B 0,C 180,E1 -25374.208,E2 -25374.208} C_VEL
LIN {X 0,Y 213.283,Z 571.236,A -85,B 0,C 180,E1 -25377.765,E2 -25377.765} C_VEL
LIN {X 0,Y 214.754,Z 574.741,A -85,B 0,C 180,E1 -25380.301,E2 -25380.301} C_VEL
LIN {X 0,Y 217.286,Z 580.777,A -85,B 0,C 180,E1 -25383.621,E2 -25383.621} C_VEL
LIN {X 0,Y 216.056,Z 592.749,A -85,B 0,C 180,E1 -25383.981,E2 -25383.981} C_VEL
LIN {X 0,Y 212.432,Z 624.655,A -85,B 0,C 180,E1 -25384.802,E2 -25384.802} C_VEL
LIN {X 0,Y 209.387,Z 640.451,A -85,B 0,C 180,E1 -25385.397,E2 -25385.397} C_VEL
LIN {X 0,Y 205.59,Z 654.514,A -85,B 0,C 180,E1 -25386.17,E2 -25386.17} C_VEL
LIN {X 0,Y 200.586,Z 668.94,A -85,B 0,C 180,E1 -25387.269,E2 -25387.269} C_VEL
LIN {X 0,Y 194.553,Z 682.911,A -85,B 0,C 180,E1 -25388.66,E2 -25388.66} C_VEL
LIN {X 0,Y 187.554,Z 696.299,A -85,B 0,C 180,E1 -25390.39,E2 -25390.39} C_VEL
LIN {X 0,Y 179.946,Z 708.637,A -85,B 0,C 180,E1 -25392.48,E2 -25392.48} C_VEL
LIN {X 0,Y 172.612,Z 718.981,A -85,B 0,C 180,E1 -25394.77,E2 -25394.77} C_VEL
LIN {X 0,Y 164.094,Z 729.552,A -85,B 0,C 180,E1 -25397.795,E2 -25397.795} C_VEL
LIN {X 0,Y 156.212,Z 738.25,A -85,B 0,C 180,E1 -25401.096,E2 -25401.096} C_VEL
LIN {X 0,Y 147.787,Z 746.599,A -85,B 0,C 180,E1 -25405.341,E2 -25405.341} C_VEL
LIN {X 0,Y 140.063,Z 753.446,A -85,B 0,C 180,E1 -25410.118,E2 -25410.118} C_VEL
LIN {X 0,Y 133.515,Z 758.795,A -85,B 0,C 180,E1 -25415.383,E2 -25415.383} C_VEL
LIN {X 0,Y 128.074,Z 762.907,A -85,B 0,C 180,E1 -25421.186,E2 -25421.186} C_VEL
LIN {X 0,Y 123.765,Z 765.87,A -85,B 0,C 180,E1 -25427.58,E2 -25427.58} C_VEL
LIN {X 0,Y 120.825,Z 767.639,A -85,B 0,C 180,E1 -25434.523,E2 -25434.523} C_VEL
LIN {X 0,Y 119.114,Z 768.144,A -85,B 0,C 180,E1 -25441.837,E2 -25441.837} C_VEL
LIN {X 0,Y 118.711,Z 767.332,A -85,B 0,C 180,E1 -25449.196,E2 -25449.196} C_VEL
LIN {X 0,Y 118.933,Z 766.441,A -85,B 0,C 180,E1 -25452.817,E2 -25452.817} C_VEL
LIN {X 0,Y 120.156,Z 763.695,A -85,B 0,C 180,E1 -25459.896,E2 -25459.896} C_VEL
LIN {X 0,Y 122.492,Z 759.647,A -85,B 0,C 180,E1 -25466.713,E2 -25466.713} C_VEL
LIN {X 0,Y 126.041,Z 754.236,A -85,B 0,C 180,E1 -25473.198,E2 -25473.198} C_VEL
LIN {X 0,Y 130.864,Z 747.319,A -85,B 0,C 180,E1 -25479.273,E2 -25479.273} C_VEL
LIN {X 0,Y 135.994,Z 739.849,A -85,B 0,C 180,E1 -25484.211,E2 -25484.211} C_VEL
LIN {X 0,Y 142.081,Z 730.834,A -85,B 0,C 180,E1 -25488.756,E2 -25488.756} C_VEL
LIN {X 0,Y 147.796,Z 721.671,A -85,B 0,C 180,E1 -25492.361,E2 -25492.361} C_VEL
LIN {X 0,Y 154.084,Z 710.815,A -85,B 0,C 180,E1 -25495.679,E2 -25495.679} C_VEL
LIN {X 0,Y 160.225,Z 698.971,A -85,B 0,C 180,E1 -25498.488,E2 -25498.488} C_VEL
LIN {X 0,Y 166.093,Z 686.024,A -85,B 0,C 180,E1 -25500.868,E2 -25500.868} C_VEL
LIN {X 0,Y 171.463,Z 671.845,A -85,B 0,C 180,E1 -25502.896,E2 -25502.896} C_VEL
LIN {X 0,Y 176.132,Z 656.919,A -85,B 0,C 180,E1 -25504.48,E2 -25504.48} C_VEL
LIN {X 0,Y 179.705,Z 642.071,A -85,B 0,C 180,E1 -25505.66,E2 -25505.66} C_VEL
LIN {X 0,Y 182.469,Z 626.657,A -85,B 0,C 180,E1 -25506.487,E2 -25506.487} C_VEL
LIN {X 0,Y 184.655,Z 606.359,A -85,B 0,C 180,E1 -25507.178,E2 -25507.178} C_VEL
LIN {X 0,Y 188.448,Z 564.156,A -85,B 0,C 180,E1 -25508.447,E2 -25508.447} C_VEL
LIN {X 0,Y 183.429,Z 554.122,A -85,B 0,C 180,E1 -25511.405,E2 -25511.405} C_VEL
LIN {X 0,Y 177.732,Z 543.782,A -85,B 0,C 180,E1 -25515.162,E2 -25515.162} C_VEL
LIN {X 0,Y 173.243,Z 536.41,A -85,B 0,C 180,E1 -25518.545,E2 -25518.545} C_VEL
LIN {X 0,Y 169.171,Z 530.082,A -85,B 0,C 180,E1 -25522.058,E2 -25522.058} C_VEL
LIN {X 0,Y 166.08,Z 525.523,A -85,B 0,C 180,E1 -25525.153,E2 -25525.153} C_VEL
LIN {X 0,Y 163.505,Z 521.777,A -85,B 0,C 180,E1 -25528.154,E2 -25528.154} C_VEL
LIN {X 0,Y 160.936,Z 518.035,A -85,B 0,C 180,E1 -25531.756,E2 -25531.756} C_VEL
LIN {X 0,Y 160.411,Z 517.281,A -85,B 0,C 180,E1 -25532.597,E2 -25532.597} C_VEL
LIN {X 0,Y 158.112,Z 514.675,A -85,B 0,C 180,E1 -25536.903,E2 -25536.903} C_VEL
LIN {X 0,Y 157.19,Z 512.421,A -85,B 0,C 180,E1 -25539.557,E2 -25539.557} C_VEL
LIN {X 0,Y 155.562,Z 511.156,A -85,B 0,C 180,E1 -25549.588,E2 -25549.588} C_VEL
LIN {X 0,Y 157.545,Z 512.264,A -85,B 0,C 180,E1 -25558.824,E2 -25558.824} C_VEL
LIN {X 0,Y 158.902,Z 515.33,A -85,B 0,C 180,E1 -25562.274,E2 -25562.274} C_VEL
LIN {X 0,Y 160.964,Z 517.601,A -85,B 0,C 180,E1 -25565.789,E2 -25565.789} C_VEL
LIN {X 0,Y 163.415,Z 521.416,A -85,B 0,C 180,E1 -25569.28,E2 -25569.28} C_VEL
LIN {X 0,Y 164.641,Z 523.155,A -85,B 0,C 180,E1 -25570.779,E2 -25570.779} C_VEL
LIN {X 0,Y 167.23,Z 526.998,A -85,B 0,C 180,E1 -25573.596,E2 -25573.596} C_VEL
LIN {X 0,Y 170.315,Z 531.78,A -85,B 0,C 180,E1 -25576.566,E2 -25576.566} C_VEL
LIN {X 0,Y 173.339,Z 536.474,A -85,B 0,C 180,E1 -25579.099,E2 -25579.099} C_VEL
LIN {X 0,Y 178.341,Z 544.817,A -85,B 0,C 180,E1 -25582.843,E2 -25582.843} C_VEL
LIN {X 0,Y 183.141,Z 555.697,A -85,B 0,C 180,E1 -25586.158,E2 -25586.158} C_VEL
LIN {X 0,Y 187.598,Z 567.018,A -85,B 0,C 180,E1 -25588.972,E2 -25588.972} C_VEL
LIN {X 0,Y 188.216,Z 568.721,A -85,B 0,C 180,E1 -25589.346,E2 -25589.346} C_VEL
LIN {X 0,Y 182.704,Z 629.202,A -85,B 0,C 180,E1 -25591.223,E2 -25591.223} C_VEL
LIN {X 0,Y 180.181,Z 644.801,A -85,B 0,C 180,E1 -25591.965,E2 -25591.965} C_VEL
LIN {X 0,Y 176.505,Z 660.195,A -85,B 0,C 180,E1 -25593,E2 -25593} C_VEL
LIN {X 0,Y 172.304,Z 674.055,A -85,B 0,C 180,E1 -25594.313,E2 -25594.313} C_VEL
LIN {X 0,Y 167.016,Z 688.277,A -85,B 0,C 180,E1 -25596.094,E2 -25596.094} C_VEL
LIN {X 0,Y 161.765,Z 700.229,A -85,B 0,C 180,E1 -25598.05,E2 -25598.05} C_VEL
LIN {X 0,Y 155.935,Z 711.912,A -85,B 0,C 180,E1 -25600.485,E2 -25600.485} C_VEL
LIN {X 0,Y 149.91,Z 722.78,A -85,B 0,C 180,E1 -25603.391,E2 -25603.391} C_VEL
LIN {X 0,Y 143.782,Z 732.814,A -85,B 0,C 180,E1 -25606.817,E2 -25606.817} C_VEL
LIN {X 0,Y 138.33,Z 741.378,A -85,B 0,C 180,E1 -25610.573,E2 -25610.573} C_VEL
LIN {X 0,Y 132.662,Z 749.743,A -85,B 0,C 180,E1 -25615.283,E2 -25615.283} C_VEL
LIN {X 0,Y 127.915,Z 756.631,A -85,B 0,C 180,E1 -25620.363,E2 -25620.363} C_VEL
LIN {X 0,Y 123.765,Z 762.997,A -85,B 0,C 180,E1 -25626.577,E2 -25626.577} C_VEL
LIN {X 0,Y 122.93,Z 764.355,A -85,B 0,C 180,E1 -25628.186,E2 -25628.186} C_VEL
LIN {X 0,Y 121.181,Z 766.318,A -85,B 0,C 180,E1 -25630.681,E2 -25630.681} C_VEL
LIN {X 0,Y 116.921,Z 768.974,A -85,B 0,C 180,E1 -25634.799,E2 -25634.799} C_VEL
LIN {X 0,Y 113.735,Z 770.733,A -85,B 0,C 180,E1 -25638.327,E2 -25638.327} C_VEL
LIN {X 0,Y 112.264,Z 772.067,A -85,B 0,C 180,E1 -25641.688,E2 -25641.688} C_VEL
LIN {X 0,Y 112.216,Z 772.187,A -85,B 0,C 180,E1 -25642.183,E2 -25642.183} C_VEL
LIN {X 0,Y 112.118,Z 773.446,A -85,B 0,C 180,E1 -25646.404,E2 -25646.404} C_VEL
LIN {X 0,Y 112.258,Z 774.175,A -85,B 0,C 180,E1 -25649.998,E2 -25649.998} C_VEL
LIN {X 0,Y 112.139,Z 774.706,A -85,B 0,C 180,E1 -25657.199,E2 -25657.199} C_VEL
LIN {X 0,Y 113.16,Z 774.067,A -85,B 0,C 180,E1 -25664.382,E2 -25664.382} C_VEL
LIN {X 0,Y 115.615,Z 772.332,A -85,B 0,C 180,E1 -25671.389,E2 -25671.389} C_VEL
LIN {X 0,Y 119.676,Z 769.372,A -85,B 0,C 180,E1 -25678.254,E2 -25678.254} C_VEL
LIN {X 0,Y 125.044,Z 765.468,A -85,B 0,C 180,E1 -25684.194,E2 -25684.194} C_VEL
LIN {X 0,Y 131.796,Z 760.143,A -85,B 0,C 180,E1 -25689.782,E2 -25689.782} C_VEL
LIN {X 0,Y 139.76,Z 753.416,A -85,B 0,C 180,E1 -25694.746,E2 -25694.746} C_VEL
LIN {X 0,Y 148.547,Z 745.147,A -85,B 0,C 180,E1 -25699.196,E2 -25699.196} C_VEL
LIN {X 0,Y 157.06,Z 736.384,A -85,B 0,C 180,E1 -25702.582,E2 -25702.582} C_VEL
LIN {X 0,Y 166.101,Z 725.919,A -85,B 0,C 180,E1 -25705.593,E2 -25705.593} C_VEL
LIN {X 0,Y 172.762,Z 717.167,A -85,B 0,C 180,E1 -25707.574,E2 -25707.574} C_VEL
LIN {X 0,Y 180.91,Z 705.061,A -85,B 0,C 180,E1 -25709.696,E2 -25709.696} C_VEL
LIN {X 0,Y 188.208,Z 692.538,A -85,B 0,C 180,E1 -25711.342,E2 -25711.342} C_VEL
LIN {X 0,Y 194.769,Z 679.184,A -85,B 0,C 180,E1 -25712.69,E2 -25712.69} C_VEL
LIN {X 0,Y 200.37,Z 665.45,A -85,B 0,C 180,E1 -25713.712,E2 -25713.712} C_VEL
LIN {X 0,Y 205.263,Z 650.126,A -85,B 0,C 180,E1 -25714.558,E2 -25714.558} C_VEL
LIN {X 0,Y 208.852,Z 634.767,A -85,B 0,C 180,E1 -25715.16,E2 -25715.16} C_VEL
LIN {X 0,Y 211.297,Z 618.26,A -85,B 0,C 180,E1 -25715.61,E2 -25715.61} C_VEL
LIN {X 0,Y 214.727,Z 587.22,A -85,B 0,C 180,E1 -25716.385,E2 -25716.385} C_VEL
LIN {X 0,Y 213.357,Z 582.189,A -85,B 0,C 180,E1 -25718.63,E2 -25718.63} C_VEL
LIN {X 0,Y 212.484,Z 579.616,A -85,B 0,C 180,E1 -25720.234,E2 -25720.234} C_VEL
LIN {X 0,Y 211.597,Z 577.477,A -85,B 0,C 180,E1 -25722.135,E2 -25722.135} C_VEL
LIN {X 0,Y 210.532,Z 574.341,A -85,B 0,C 180,E1 -25725.846,E2 -25725.846} C_VEL
LIN {X 0,Y 210.207,Z 573.953,A -85,B 0,C 180,E1 -25730.377,E2 -25730.377} C_VEL
LIN {X 0,Y 210.865,Z 574.637,A -85,B 0,C 180,E1 -25733.853,E2 -25733.853} C_VEL
LIN {X 0,Y 212.041,Z 577.952,A -85,B 0,C 180,E1 -25737.229,E2 -25737.229} C_VEL
LIN {X 0,Y 213.341,Z 581.271,A -85,B 0,C 180,E1 -25739.659,E2 -25739.659} C_VEL
LIN {X 0,Y 214.882,Z 585.259,A -85,B 0,C 180,E1 -25741.972,E2 -25741.972} C_VEL
LIN {X 0,Y 210.255,Z 625.218,A -85,B 0,C 180,E1 -25742.978,E2 -25742.978} C_VEL
LIN {X 0,Y 207.105,Z 641.021,A -85,B 0,C 180,E1 -25743.554,E2 -25743.554} C_VEL
LIN {X 0,Y 203.067,Z 655.477,A -85,B 0,C 180,E1 -25744.328,E2 -25744.328} C_VEL
LIN {X 0,Y 197.668,Z 670.331,A -85,B 0,C 180,E1 -25745.439,E2 -25745.439} C_VEL
LIN {X 0,Y 191.12,Z 684.714,A -85,B 0,C 180,E1 -25746.865,E2 -25746.865} C_VEL
LIN {X 0,Y 184.015,Z 697.653,A -85,B 0,C 180,E1 -25748.542,E2 -25748.542} C_VEL
LIN {X 0,Y 176.07,Z 709.939,A -85,B 0,C 180,E1 -25750.613,E2 -25750.613} C_VEL
LIN {X 0,Y 167.766,Z 721.081,A -85,B 0,C 180,E1 -25753.107,E2 -25753.107} C_VEL
LIN {X 0,Y 159.079,Z 731.219,A -85,B 0,C 180,E1 -25756.083,E2 -25756.083} C_VEL
LIN {X 0,Y 150.848,Z 739.757,A -85,B 0,C 180,E1 -25759.43,E2 -25759.43} C_VEL
LIN {X 0,Y 143.256,Z 746.791,A -85,B 0,C 180,E1 -25763.109,E2 -25763.109} C_VEL
LIN {X 0,Y 135.066,Z 753.647,A -85,B 0,C 180,E1 -25767.925,E2 -25767.925} C_VEL
LIN {X 0,Y 128.019,Z 759.015,A -85,B 0,C 180,E1 -25773.298,E2 -25773.298} C_VEL
LIN {X 0,Y 122.082,Z 763.13,A -85,B 0,C 180,E1 -25779.291,E2 -25779.291} C_VEL
LIN {X 0,Y 117.358,Z 766.079,A -85,B 0,C 180,E1 -25785.942,E2 -25785.942} C_VEL
LIN {X 0,Y 114.105,Z 767.845,A -85,B 0,C 180,E1 -25793.199,E2 -25793.199} C_VEL
LIN {X 0,Y 112.087,Z 768.337,A -85,B 0,C 180,E1 -25801.382,E2 -25801.382} C_VEL
LIN {X 0,Y 111.591,Z 767.708,A -85,B 0,C 180,E1 -25807.8,E2 -25807.8} C_VEL
LIN {X 0,Y 111.77,Z 766.893,A -85,B 0,C 180,E1 -25811.678,E2 -25811.678} C_VEL
LIN {X 0,Y 112.837,Z 764.319,A -85,B 0,C 180,E1 -25819.233,E2 -25819.233} C_VEL
LIN {X 0,Y 115.161,Z 760.453,A -85,B 0,C 180,E1 -25826.503,E2 -25826.503} C_VEL
LIN {X 0,Y 118.771,Z 755.231,A -85,B 0,C 180,E1 -25833.394,E2 -25833.394} C_VEL
LIN {X 0,Y 123.693,Z 748.522,A -85,B 0,C 180,E1 -25839.816,E2 -25839.816} C_VEL
LIN {X 0,Y 129.016,Z 741.27,A -85,B 0,C 180,E1 -25844.998,E2 -25844.998} C_VEL
LIN {X 0,Y 135.277,Z 732.503,A -85,B 0,C 180,E1 -25849.741,E2 -25849.741} C_VEL
LIN {X 0,Y 142.175,Z 721.98,A -85,B 0,C 180,E1 -25854.069,E2 -25854.069} C_VEL
LIN {X 0,Y 148.747,Z 711.133,A -85,B 0,C 180,E1 -25857.432,E2 -25857.432} C_VEL
LIN {X 0,Y 155.116,Z 699.306,A -85,B 0,C 180,E1 -25860.27,E2 -25860.27} C_VEL
LIN {X 0,Y 161.196,Z 686.395,A -85,B 0,C 180,E1 -25862.654,E2 -25862.654} C_VEL
LIN {X 0,Y 166.739,Z 672.261,A -85,B 0,C 180,E1 -25864.683,E2 -25864.683} C_VEL
LIN {X 0,Y 171.561,Z 657.391,A -85,B 0,C 180,E1 -25866.26,E2 -25866.26} C_VEL
LIN {X 0,Y 175.242,Z 642.641,A -85,B 0,C 180,E1 -25867.434,E2 -25867.434} C_VEL
LIN {X 0,Y 178.093,Z 627.418,A -85,B 0,C 180,E1 -25868.249,E2 -25868.249} C_VEL
LIN {X 0,Y 180.102,Z 610.076,A -85,B 0,C 180,E1 -25868.854,E2 -25868.854} C_VEL
LIN {X 0,Y 184.098,Z 567.213,A -85,B 0,C 180,E1 -25870.129,E2 -25870.129} C_VEL
LIN {X 0,Y 179.873,Z 558.505,A -85,B 0,C 180,E1 -25872.829,E2 -25872.829} C_VEL
LIN {X 0,Y 174.786,Z 549.108,A -85,B 0,C 180,E1 -25876.404,E2 -25876.404} C_VEL
LIN {X 0,Y 170.447,Z 541.694,A -85,B 0,C 180,E1 -25879.896,E2 -25879.896} C_VEL
LIN {X 0,Y 166.451,Z 535.365,A -85,B 0,C 180,E1 -25883.647,E2 -25883.647} C_VEL
LIN {X 0,Y 164.379,Z 532.109,A -85,B 0,C 180,E1 -25885.858,E2 -25885.858} C_VEL
LIN {X 0,Y 161.855,Z 528.321,A -85,B 0,C 180,E1 -25888.974,E2 -25888.974} C_VEL
LIN {X 0,Y 159.396,Z 524.501,A -85,B 0,C 180,E1 -25892.648,E2 -25892.648} C_VEL
LIN {X 0,Y 156.778,Z 521.195,A -85,B 0,C 180,E1 -25897.825,E2 -25897.825} C_VEL
LIN {X 0,Y 156.116,Z 519.369,A -85,B 0,C 180,E1 -25899.954,E2 -25899.954} C_VEL
LIN {X 0,Y 154.636,Z 518.203,A -85,B 0,C 180,E1 -25909.525,E2 -25909.525} C_VEL
LIN {X 0,Y 156.407,Z 519.235,A -85,B 0,C 180,E1 -25918.324,E2 -25918.324} C_VEL
LIN {X 0,Y 157.945,Z 522.555,A -85,B 0,C 180,E1 -25922.288,E2 -25922.288} C_VEL
LIN {X 0,Y 159.51,Z 524.284,A -85,B 0,C 180,E1 -25925.055,E2 -25925.055} C_VEL
LIN {X 0,Y 162.082,Z 528.306,A -85,B 0,C 180,E1 -25928.863,E2 -25928.863} C_VEL
LIN {X 0,Y 165.198,Z 533.138,A -85,B 0,C 180,E1 -25932.593,E2 -25932.593} C_VEL
LIN {X 0,Y 168.858,Z 539.042,A -85,B 0,C 180,E1 -25936.263,E2 -25936.263} C_VEL
LIN {X 0,Y 173.539,Z 546.787,A -85,B 0,C 180,E1 -25940.202,E2 -25940.202} C_VEL
LIN {X 0,Y 176.146,Z 551.754,A -85,B 0,C 180,E1 -25942.203,E2 -25942.203} C_VEL
LIN {X 0,Y 180.783,Z 562.94,A -85,B 0,C 180,E1 -25945.557,E2 -25945.557} C_VEL
LIN {X 0,Y 183.887,Z 571.245,A -85,B 0,C 180,E1 -25947.646,E2 -25947.646} C_VEL
LIN {X 0,Y 178.332,Z 629.692,A -85,B 0,C 180,E1 -25949.451,E2 -25949.451} C_VEL
LIN {X 0,Y 175.625,Z 645.554,A -85,B 0,C 180,E1 -25950.217,E2 -25950.217} C_VEL
LIN {X 0,Y 172.018,Z 660.106,A -85,B 0,C 180,E1 -25951.192,E2 -25951.192} C_VEL
LIN {X 0,Y 167.69,Z 673.946,A -85,B 0,C 180,E1 -25952.492,E2 -25952.492} C_VEL
